LIN {X 0,Y 284.126,Z 570.884,A -85,B 0,C 180,E1 -16986.134,E2 -16986.134} C_VEL
LIN {X 0,Y 285.514,Z 585.301,A -85,B 0,C 180,E1 -16986.902,E2 -16986.902} C_VEL
LIN {X 0,Y 286.444,Z 597.974,A -85,B 0,C 180,E1 -16987.838,E2 -16987.838} C_VEL
LIN {X 0,Y 287.043,Z 610.993,A -85,B 0,C 180,E1 -16989.097,E2 -16989.097} C_VEL
LIN {X 0,Y 287.237,Z 622.835,A -85,B 0,C 180,E1 -16990.527,E2 -16990.527} C_VEL
LIN {X 0,Y 286.97,Z 632.757,A -85,B 0,C 180,E1 -16991.99,E2 -16991.99} C_VEL
LIN {X 0,Y 285.776,Z 641.656,A -85,B 0,C 180,E1 -16993.56,E2 -16993.56} C_VEL
LIN {X 0,Y 284.464,Z 651.441,A -85,B 0,C 180,E1 -16995.696,E2 -16995.696} C_VEL
LIN {X 0,Y 283.789,Z 659.297,A -85,B 0,C 180,E1 -16997.848,E2 -16997.848} C_VEL
LIN {X 0,Y 283.448,Z 665.562,A -85,B 0,C 180,E1 -17000.005,E2 -17000.005} C_VEL
LIN {X 0,Y 283.441,Z 670.658,A -85,B 0,C 180,E1 -17002.234,E2 -17002.234} C_VEL
LIN {X 0,Y 283.67,Z 674.283,A -85,B 0,C 180,E1 -17004.313,E2 -17004.313} C_VEL
LIN {X 0,Y 283.832,Z 676.171,A -85,B 0,C 180,E1 -17005.74,E2 -17005.74} C_VEL
LIN {X 0,Y 283.974,Z 677.598,A -85,B 0,C 180,E1 -17007.163,E2 -17007.163} C_VEL
LIN {X 0,Y 284.233,Z 678.549,A -85,B 0,C 180,E1 -17008.583,E2 -17008.583} C_VEL
LIN {X 0,Y 284.459,Z 679.061,A -85,B 0,C 180,E1 -17010,E2 -17010} C_VEL
LIN {X 0,Y 283.861,Z 678.655,A -85,B 0,C 180,E1 -17012.838,E2 -17012.838} C_VEL
LIN {X 0,Y 283.692,Z 677.798,A -85,B 0,C 180,E1 -17014.262,E2 -17014.262} C_VEL
LIN {X 0,Y 283.264,Z 674.815,A -85,B 0,C 180,E1 -17017.126,E2 -17017.126} C_VEL
LIN {X 0,Y 283.136,Z 671.429,A -85,B 0,C 180,E1 -17019.285,E2 -17019.285} C_VEL
LIN {X 0,Y 283.389,Z 667.023,A -85,B 0,C 180,E1 -17021.444,E2 -17021.444} C_VEL
LIN {X 0,Y 284.212,Z 660.522,A -85,B 0,C 180,E1 -17023.952,E2 -17023.952} C_VEL
LIN {X 0,Y 285.074,Z 654.806,A -85,B 0,C 180,E1 -17025.735,E2 -17025.735} C_VEL
LIN {X 0,Y 286.836,Z 646.656,A -85,B 0,C 180,E1 -17027.835,E2 -17027.835} C_VEL
LIN {X 0,Y 289.074,Z 636.649,A -85,B 0,C 180,E1 -17029.9,E2 -17029.9} C_VEL
LIN {X 0,Y 290.359,Z 625.448,A -85,B 0,C 180,E1 -17031.848,E2 -17031.848} C_VEL
LIN {X 0,Y 291.533,Z 612.796,A -85,B 0,C 180,E1 -17033.642,E2 -17033.642} C_VEL
LIN {X 0,Y 291.696,Z 600.649,A -85,B 0,C 180,E1 -17035.122,E2 -17035.122} C_VEL
LIN {X 0,Y 290.667,Z 587.531,A -85,B 0,C 180,E1 -17036.541,E2 -17036.541} C_VEL
LIN {X 0,Y 288.705,Z 574.355,A -85,B 0,C 180,E1 -17037.828,E2 -17037.828} C_VEL
LIN {X 0,Y 286.15,Z 563.427,A -85,B 0,C 180,E1 -17038.838,E2 -17038.838} C_VEL
LIN {X 0,Y 285.515,Z 560.161,A -85,B 0,C 180,E1 -17039.106,E2 -17039.106} C_VEL
LIN {X 0,Y 287.109,Z 549.67,A -85,B 0,C 180,E1 -17043.667,E2 -17043.667} C_VEL
LIN {X 0,Y 289.085,Z 539.77,A -85,B 0,C 180,E1 -17048.193,E2 -17048.193} C_VEL
LIN {X 0,Y 289.175,Z 537.775,A -85,B 0,C 180,E1 -17049.191,E2 -17049.191} C_VEL
LIN {X 0,Y 288.339,Z 532.571,A -85,B 0,C 180,E1 -17052.035,E2 -17052.035} C_VEL
LIN {X 0,Y 287.355,Z 527.335,A -85,B 0,C 180,E1 -17055.176,E2 -17055.176} C_VEL
LIN {X 0,Y 286.33,Z 522.347,A -85,B 0,C 180,E1 -17058.493,E2 -17058.493} C_VEL
LIN {X 0,Y 285.335,Z 517.677,A -85,B 0,C 180,E1 -17062.017,E2 -17062.017} C_VEL
LIN {X 0,Y 284.314,Z 513.065,A -85,B 0,C 180,E1 -17066.208,E2 -17066.208} C_VEL
LIN {X 0,Y 284.361,Z 513.057,A -85,B 0,C 180,E1 -17070.377,E2 -17070.377} C_VEL
LIN {X 0,Y 284.381,Z 513.053,A -85,B 0,C 180,E1 -17073.587,E2 -17073.587} C_VEL
LIN {X 0,Y 284.369,Z 513.056,A -85,B 0,C 180,E1 -17076.707,E2 -17076.707} C_VEL
LIN {X 0,Y 284.406,Z 513.055,A -85,B 0,C 180,E1 -17081.262,E2 -17081.262} C_VEL
LIN {X 0,Y 284.495,Z 513.044,A -85,B 0,C 180,E1 -17084.459,E2 -17084.459} C_VEL
LIN {X 0,Y 284.492,Z 513.04,A -85,B 0,C 180,E1 -17088.602,E2 -17088.602} C_VEL
LIN {X 0,Y 284.663,Z 513.019,A -85,B 0,C 180,E1 -17091.482,E2 -17091.482} C_VEL
LIN {X 0,Y 284.6,Z 513.031,A -85,B 0,C 180,E1 -17094.332,E2 -17094.332} C_VEL
LIN {X 0,Y 284.854,Z 513.002,A -85,B 0,C 180,E1 -17098.587,E2 -17098.587} C_VEL
LIN {X 0,Y 284.858,Z 513.003,A -85,B 0,C 180,E1 -17101.414,E2 -17101.414} C_VEL
LIN {X 0,Y 284.582,Z 513.031,A -85,B 0,C 180,E1 -17105.536,E2 -17105.536} C_VEL
LIN {X 0,Y 285.22,Z 515.176,A -85,B 0,C 180,E1 -17105.834,E2 -17105.834} C_VEL
LIN {X 0,Y 288.767,Z 521.378,A -85,B 0,C 180,E1 -17106.99,E2 -17106.99} C_VEL
LIN {X 0,Y 293.537,Z 532.381,A -85,B 0,C 180,E1 -17108.954,E2 -17108.954} C_VEL
LIN {X 0,Y 296.554,Z 541.172,A -85,B 0,C 180,E1 -17110.584,E2 -17110.584} C_VEL
LIN {X 0,Y 298.373,Z 548.706,A -85,B 0,C 180,E1 -17112.039,E2 -17112.039} C_VEL
LIN {X 0,Y 297.747,Z 553.329,A -85,B 0,C 180,E1 -17112.77,E2 -17112.77} C_VEL
LIN {X 0,Y 295.774,Z 562.817,A -85,B 0,C 180,E1 -17114.447,E2 -17114.447} C_VEL
LIN {X 0,Y 293.677,Z 571.656,A -85,B 0,C 180,E1 -17116.417,E2 -17116.417} C_VEL
LIN {X 0,Y 291.671,Z 579.309,A -85,B 0,C 180,E1 -17118.563,E2 -17118.563} C_VEL
LIN {X 0,Y 290.018,Z 584.973,A -85,B 0,C 180,E1 -17120.572,E2 -17120.572} C_VEL
LIN {X 0,Y 288.412,Z 590.115,A -85,B 0,C 180,E1 -17122.948,E2 -17122.948} C_VEL
LIN {X 0,Y 287.211,Z 593.585,A -85,B 0,C 180,E1 -17125.124,E2 -17125.124} C_VEL
LIN {X 0,Y 286.03,Z 596.426,A -85,B 0,C 180,E1 -17127.83,E2 -17127.83} C_VEL
LIN {X 0,Y 285.27,Z 597.703,A -85,B 0,C 180,E1 -17130.427,E2 -17130.427} C_VEL
LIN {X 0,Y 284.803,Z 597.654,A -85,B 0,C 180,E1 -17132.964,E2 -17132.964} C_VEL
LIN {X 0,Y 284.628,Z 596.402,A -85,B 0,C 180,E1 -17135.429,E2 -17135.429} C_VEL
LIN {X 0,Y 284.722,Z 593.682,A -85,B 0,C 180,E1 -17138.105,E2 -17138.105} C_VEL
LIN {X 0,Y 285.201,Z 589.25,A -85,B 0,C 180,E1 -17140.843,E2 -17140.843} C_VEL
LIN {X 0,Y 285.807,Z 584.791,A -85,B 0,C 180,E1 -17142.886,E2 -17142.886} C_VEL
LIN {X 0,Y 286.656,Z 578.043,A -85,B 0,C 180,E1 -17145.317,E2 -17145.317} C_VEL
LIN {X 0,Y 287.491,Z 571.602,A -85,B 0,C 180,E1 -17147.171,E2 -17147.171} C_VEL
LIN {X 0,Y 288.739,Z 562.674,A -85,B 0,C 180,E1 -17149.253,E2 -17149.253} C_VEL
LIN {X 0,Y 289.919,Z 552.701,A -85,B 0,C 180,E1 -17151.147,E2 -17151.147} C_VEL
LIN {X 0,Y 291.151,Z 541.755,A -85,B 0,C 180,E1 -17152.806,E2 -17152.806} C_VEL
LIN {X 0,Y 291.404,Z 537.676,A -85,B 0,C 180,E1 -17153.35,E2 -17153.35} C_VEL
LIN {X 0,Y 288.411,Z 526.574,A -85,B 0,C 180,E1 -17154.868,E2 -17154.868} C_VEL
LIN {X 0,Y 284.684,Z 514.526,A -85,B 0,C 180,E1 -17156.257,E2 -17156.257} C_VEL
LIN {X 0,Y 284.32,Z 513.07,A -85,B 0,C 180,E1 -17156.421,E2 -17156.421} C_VEL
LIN {X 0,Y 284.364,Z 513.063,A -85,B 0,C 180,E1 -17160.376,E2 -17160.376} C_VEL
LIN {X 0,Y 284.385,Z 513.062,A -85,B 0,C 180,E1 -17163.587,E2 -17163.587} C_VEL
LIN {X 0,Y 284.337,Z 513.065,A -85,B 0,C 180,E1 -17166.704,E2 -17166.704} C_VEL
LIN {X 0,Y 284.381,Z 513.06,A -85,B 0,C 180,E1 -17169.904,E2 -17169.904} C_VEL
LIN {X 0,Y 284.452,Z 513.05,A -85,B 0,C 180,E1 -17174.492,E2 -17174.492} C_VEL
LIN {X 0,Y 284.488,Z 513.046,A -85,B 0,C 180,E1 -17178.601,E2 -17178.601} C_VEL
LIN {X 0,Y 284.613,Z 513.033,A -85,B 0,C 180,E1 -17181.48,E2 -17181.48} C_VEL
LIN {X 0,Y 284.581,Z 513.034,A -85,B 0,C 180,E1 -17184.331,E2 -17184.331} C_VEL
LIN {X 0,Y 284.855,Z 513,A -85,B 0,C 180,E1 -17188.586,E2 -17188.586} C_VEL
LIN {X 0,Y 284.857,Z 513.003,A -85,B 0,C 180,E1 -17191.414,E2 -17191.414} C_VEL
LIN {X 0,Y 284.648,Z 513.029,A -85,B 0,C 180,E1 -17197.091,E2 -17197.091} C_VEL
LIN {X 0,Y 284.518,Z 513.041,A -85,B 0,C 180,E1 -17199.957,E2 -17199.957} C_VEL
LIN {X 0,Y 284.468,Z 513.048,A -85,B 0,C 180,E1 -17204.303,E2 -17204.303} C_VEL
LIN {X 0,Y 284.39,Z 513.058,A -85,B 0,C 180,E1 -17208.739,E2 -17208.739} C_VEL
LIN {X 0,Y 284.33,Z 513.066,A -85,B 0,C 180,E1 -17211.763,E2 -17211.763} C_VEL
LIN {X 0,Y 284.32,Z 513.068,A -85,B 0,C 180,E1 -17214.848,E2 -17214.848} C_VEL
LIN {X 0,Y 284.295,Z 513.069,A -85,B 0,C 180,E1 -17218.014,E2 -17218.014} C_VEL
LIN {X 0,Y 284.29,Z 513.074,A -85,B 0,C 180,E1 -17221.275,E2 -17221.275} C_VEL
LIN {X 0,Y 284.339,Z 513.066,A -85,B 0,C 180,E1 -17225.346,E2 -17225.346} C_VEL
LIN {X 0,Y 284.304,Z 513.068,A -85,B 0,C 180,E1 -17228.17,E2 -17228.17} C_VEL
LIN {X 0,Y 284.24,Z 513.075,A -85,B 0,C 180,E1 -17232.117,E2 -17232.117} C_VEL
LIN {X 0,Y 284.257,Z 513.074,A -85,B 0,C 180,E1 -17236.189,E2 -17236.189} C_VEL
LIN {X 0,Y 284.309,Z 513.067,A -85,B 0,C 180,E1 -17240.024,E2 -17240.024} C_VEL
LIN {X 0,Y 284.333,Z 513.065,A -85,B 0,C 180,E1 -17243.613,E2 -17243.613} C_VEL
LIN {X 0,Y 284.31,Z 513.071,A -85,B 0,C 180,E1 -17247.189,E2 -17247.189} C_VEL
LIN {X 0,Y 284.361,Z 513.06,A -85,B 0,C 180,E1 -17250.376,E2 -17250.376} C_VEL
LIN {X 0,Y 284.38,Z 513.06,A -85,B 0,C 180,E1 -17253.586,E2 -17253.586} C_VEL
LIN {X 0,Y 284.335,Z 513.067,A -85,B 0,C 180,E1 -17256.704,E2 -17256.704} C_VEL
LIN {X 0,Y 284.406,Z 513.058,A -85,B 0,C 180,E1 -17261.261,E2 -17261.261} C_VEL
LIN {X 0,Y 284.494,Z 513.046,A -85,B 0,C 180,E1 -17264.459,E2 -17264.459} C_VEL
LIN {X 0,Y 284.485,Z 513.047,A -85,B 0,C 180,E1 -17268.601,E2 -17268.601} C_VEL
LIN {X 0,Y 284.613,Z 513.031,A -85,B 0,C 180,E1 -17271.479,E2 -17271.479} C_VEL
LIN {X 0,Y 284.58,Z 513.034,A -85,B 0,C 180,E1 -17274.33,E2 -17274.33} C_VEL
LIN {X 0,Y 284.853,Z 513.002,A -85,B 0,C 180,E1 -17278.586,E2 -17278.586} C_VEL
LIN {X 0,Y 284.853,Z 513.001,A -85,B 0,C 180,E1 -17281.413,E2 -17281.413} C_VEL
LIN {X 0,Y 284.634,Z 513.029,A -85,B 0,C 180,E1 -17287.222,E2 -17287.222} C_VEL
LIN {X 0,Y 284.519,Z 513.041,A -85,B 0,C 180,E1 -17289.957,E2 -17289.957} C_VEL
LIN {X 0,Y 284.452,Z 513.049,A -85,B 0,C 180,E1 -17293.37,E2 -17293.37} C_VEL
LIN {X 0,Y 283.765,Z 513.138,A -85,B 0,C 180,E1 -17294.551,E2 -17294.551} C_VEL
LIN {X 0,Y 280.888,Z 513.496,A -85,B 0,C 180,E1 -17296.474,E2 -17296.474} C_VEL
LIN {X 0,Y 278.45,Z 513.799,A -85,B 0,C 180,E1 -17298.036,E2 -17298.036} C_VEL
LIN {X 0,Y 277.398,Z 513.93,A -85,B 0,C 180,E1 -17299.247,E2 -17299.247} C_VEL
LIN {X 0,Y 277.308,Z 513.939,A -85,B 0,C 180,E1 -17299.657,E2 -17299.657} C_VEL
LIN {X 0,Y 277.282,Z 513.943,A -85,B 0,C 180,E1 -17304.152,E2 -17304.152} C_VEL
LIN {X 0,Y 277.274,Z 513.944,A -85,B 0,C 180,E1 -17307.484,E2 -17307.484} C_VEL
LIN {X 0,Y 277.248,Z 513.949,A -85,B 0,C 180,E1 -17310.472,E2 -17310.472} C_VEL
LIN {X 0,Y 277.247,Z 513.948,A -85,B 0,C 180,E1 -17313.896,E2 -17313.896} C_VEL
LIN {X 0,Y 277.268,Z 513.946,A -85,B 0,C 180,E1 -17317.469,E2 -17317.469} C_VEL
LIN {X 0,Y 277.302,Z 514.049,A -85,B 0,C 180,E1 -17319.647,E2 -17319.647} C_VEL
LIN {X 0,Y 278.816,Z 521.939,A -85,B 0,C 180,E1 -17323.881,E2 -17323.881} C_VEL
LIN {X 0,Y 280.369,Z 529.967,A -85,B 0,C 180,E1 -17327.953,E2 -17327.953} C_VEL
LIN {X 0,Y 281.482,Z 535.685,A -85,B 0,C 180,E1 -17330.715,E2 -17330.715} C_VEL
LIN {X 0,Y 281.516,Z 539.122,A -85,B 0,C 180,E1 -17332.293,E2 -17332.293} C_VEL
LIN {X 0,Y 279.904,Z 548.574,A -85,B 0,C 180,E1 -17336.469,E2 -17336.469} C_VEL
LIN {X 0,Y 278.223,Z 559.738,A -85,B 0,C 180,E1 -17341.318,E2 -17341.318} C_VEL
LIN {X 0,Y 277.139,Z 570.066,A -85,B 0,C 180,E1 -17345.685,E2 -17345.685} C_VEL
LIN {X 0,Y 278.508,Z 584.506,A -85,B 0,C 180,E1 -17346.483,E2 -17346.483} C_VEL
LIN {X 0,Y 279.487,Z 598.226,A -85,B 0,C 180,E1 -17347.548,E2 -17347.548} C_VEL
LIN {X 0,Y 280.052,Z 611.206,A -85,B 0,C 180,E1 -17348.858,E2 -17348.858} C_VEL
LIN {X 0,Y 280.184,Z 623.313,A -85,B 0,C 180,E1 -17350.398,E2 -17350.398} C_VEL
LIN {X 0,Y 280.017,Z 631.921,A -85,B 0,C 180,E1 -17351.716,E2 -17351.716} C_VEL
LIN {X 0,Y 278.804,Z 640.734,A -85,B 0,C 180,E1 -17353.314,E2 -17353.314} C_VEL
LIN {X 0,Y 277.518,Z 649.792,A -85,B 0,C 180,E1 -17355.331,E2 -17355.331} C_VEL
LIN {X 0,Y 276.896,Z 656.55,A -85,B 0,C 180,E1 -17357.168,E2 -17357.168} C_VEL
LIN {X 0,Y 276.492,Z 662.166,A -85,B 0,C 180,E1 -17359.01,E2 -17359.01} C_VEL
LIN {X 0,Y 276.354,Z 667.634,A -85,B 0,C 180,E1 -17361.223,E2 -17361.223} C_VEL
LIN {X 0,Y 276.507,Z 671.865,A -85,B 0,C 180,E1 -17363.432,E2 -17363.432} C_VEL
LIN {X 0,Y 276.787,Z 674.949,A -85,B 0,C 180,E1 -17365.631,E2 -17365.631} C_VEL
LIN {X 0,Y 276.937,Z 676.414,A -85,B 0,C 180,E1 -17367.091,E2 -17367.091} C_VEL
LIN {X 0,Y 277.214,Z 677.425,A -85,B 0,C 180,E1 -17368.547,E2 -17368.547} C_VEL
LIN {X 0,Y 277.441,Z 677.967,A -85,B 0,C 180,E1 -17370,E2 -17370} C_VEL
LIN {X 0,Y 276.809,Z 677.621,A -85,B 0,C 180,E1 -17372.911,E2 -17372.911} C_VEL
LIN {X 0,Y 276.606,Z 676.814,A -85,B 0,C 180,E1 -17374.372,E2 -17374.372} C_VEL
LIN {X 0,Y 276.177,Z 673.883,A -85,B 0,C 180,E1 -17377.31,E2 -17377.31} C_VEL
LIN {X 0,Y 276.078,Z 670.565,A -85,B 0,C 180,E1 -17379.525,E2 -17379.525} C_VEL
LIN {X 0,Y 276.37,Z 666.254,A -85,B 0,C 180,E1 -17381.738,E2 -17381.738} C_VEL
LIN {X 0,Y 277.265,Z 659.85,A -85,B 0,C 180,E1 -17384.309,E2 -17384.309} C_VEL
LIN {X 0,Y 278.7,Z 651.977,A -85,B 0,C 180,E1 -17386.783,E2 -17386.783} C_VEL
LIN {X 0,Y 280.714,Z 643.129,A -85,B 0,C 180,E1 -17388.994,E2 -17388.994} C_VEL
LIN {X 0,Y 282.339,Z 636.416,A -85,B 0,C 180,E1 -17390.395,E2 -17390.395} C_VEL
LIN {X 0,Y 283.731,Z 625.469,A -85,B 0,C 180,E1 -17392.386,E2 -17392.386} C_VEL
LIN {X 0,Y 284.978,Z 613.667,A -85,B 0,C 180,E1 -17394.15,E2 -17394.15} C_VEL
LIN {X 0,Y 285.253,Z 601.377,A -85,B 0,C 180,E1 -17395.737,E2 -17395.737} C_VEL
LIN {X 0,Y 284.452,Z 588.865,A -85,B 0,C 180,E1 -17397.195,E2 -17397.195} C_VEL
LIN {X 0,Y 282.831,Z 576.714,A -85,B 0,C 180,E1 -17398.47,E2 -17398.47} C_VEL
LIN {X 0,Y 279.839,Z 562.965,A -85,B 0,C 180,E1 -17399.848,E2 -17399.848} C_VEL
LIN {X 0,Y 278.851,Z 558.99,A -85,B 0,C 180,E1 -17400.218,E2 -17400.218} C_VEL
LIN {X 0,Y 278.829,Z 558.603,A -85,B 0,C 180,E1 -17400.273,E2 -17400.273} C_VEL
LIN {X 0,Y 280.69,Z 547.821,A -85,B 0,C 180,E1 -17405.162,E2 -17405.162} C_VEL
LIN {X 0,Y 282.19,Z 540.774,A -85,B 0,C 180,E1 -17408.509,E2 -17408.509} C_VEL
LIN {X 0,Y 281.944,Z 537.239,A -85,B 0,C 180,E1 -17410.399,E2 -17410.399} C_VEL
LIN {X 0,Y 280.753,Z 530.313,A -85,B 0,C 180,E1 -17414.501,E2 -17414.501} C_VEL
LIN {X 0,Y 279.61,Z 524.759,A -85,B 0,C 180,E1 -17418.236,E2 -17418.236} C_VEL
LIN {X 0,Y 278.727,Z 520.574,A -85,B 0,C 180,E1 -17421.413,E2 -17421.413} C_VEL
LIN {X 0,Y 277.959,Z 517.056,A -85,B 0,C 180,E1 -17424.441,E2 -17424.441} C_VEL
LIN {X 0,Y 277.245,Z 513.946,A -85,B 0,C 180,E1 -17427.554,E2 -17427.554} C_VEL
LIN {X 0,Y 277.274,Z 513.94,A -85,B 0,C 180,E1 -17431.211,E2 -17431.211} C_VEL
LIN {X 0,Y 277.317,Z 513.939,A -85,B 0,C 180,E1 -17434.48,E2 -17434.48} C_VEL
LIN {X 0,Y 277.288,Z 513.944,A -85,B 0,C 180,E1 -17437.655,E2 -17437.655} C_VEL
LIN {X 0,Y 277.348,Z 513.938,A -85,B 0,C 180,E1 -17440.767,E2 -17440.767} C_VEL
LIN {X 0,Y 277.438,Z 513.918,A -85,B 0,C 180,E1 -17445.326,E2 -17445.326} C_VEL
LIN {X 0,Y 277.51,Z 513.916,A -85,B 0,C 180,E1 -17449.789,E2 -17449.789} C_VEL
LIN {X 0,Y 277.657,Z 513.894,A -85,B 0,C 180,E1 -17452.73,E2 -17452.73} C_VEL
LIN {X 0,Y 277.82,Z 513.878,A -85,B 0,C 180,E1 -17458.551,E2 -17458.551} C_VEL
LIN {X 0,Y 277.824,Z 513.879,A -85,B 0,C 180,E1 -17461.45,E2 -17461.45} C_VEL
LIN {X 0,Y 277.471,Z 514.008,A -85,B 0,C 180,E1 -17464.313,E2 -17464.313} C_VEL
LIN {X 0,Y 278.396,Z 516.611,A -85,B 0,C 180,E1 -17464.707,E2 -17464.707} C_VEL
LIN {X 0,Y 279.52,Z 518.046,A -85,B 0,C 180,E1 -17465.049,E2 -17465.049} C_VEL
LIN {X 0,Y 284.001,Z 526.61,A -85,B 0,C 180,E1 -17466.715,E2 -17466.715} C_VEL
LIN {X 0,Y 287.682,Z 535.557,A -85,B 0,C 180,E1 -17468.429,E2 -17468.429} C_VEL
LIN {X 0,Y 290.745,Z 545.046,A -85,B 0,C 180,E1 -17470.303,E2 -17470.303} C_VEL
LIN {X 0,Y 292.041,Z 550.664,A -85,B 0,C 180,E1 -17471.452,E2 -17471.452} C_VEL
LIN {X 0,Y 291.793,Z 553.762,A -85,B 0,C 180,E1 -17471.99,E2 -17471.99} C_VEL
LIN {X 0,Y 289.515,Z 564.005,A -85,B 0,C 180,E1 -17473.83,E2 -17473.83} C_VEL
LIN {X 0,Y 287.235,Z 573.052,A -85,B 0,C 180,E1 -17475.894,E2 -17475.894} C_VEL
LIN {X 0,Y 285.251,Z 580.192,A -85,B 0,C 180,E1 -17477.938,E2 -17477.938} C_VEL
LIN {X 0,Y 283.229,Z 586.715,A -85,B 0,C 180,E1 -17480.329,E2 -17480.329} C_VEL
LIN {X 0,Y 281.664,Z 591.393,A -85,B 0,C 180,E1 -17482.598,E2 -17482.598} C_VEL
LIN {X 0,Y 280.102,Z 595.529,A -85,B 0,C 180,E1 -17485.408,E2 -17485.408} C_VEL
LIN {X 0,Y 278.932,Z 597.926,A -85,B 0,C 180,E1 -17488.131,E2 -17488.131} C_VEL
LIN {X 0,Y 278.165,Z 598.89,A -85,B 0,C 180,E1 -17490.791,E2 -17490.791} C_VEL
LIN {X 0,Y 277.756,Z 598.557,A -85,B 0,C 180,E1 -17493.384,E2 -17493.384} C_VEL
LIN {X 0,Y 277.596,Z 597.016,A -85,B 0,C 180,E1 -17495.888,E2 -17495.888} C_VEL
LIN {X 0,Y 277.699,Z 594.36,A -85,B 0,C 180,E1 -17498.32,E2 -17498.32} C_VEL
LIN {X 0,Y 278.223,Z 589.923,A -85,B 0,C 180,E1 -17501.055,E2 -17501.055} C_VEL
LIN {X 0,Y 278.934,Z 584.846,A -85,B 0,C 180,E1 -17503.364,E2 -17503.364} C_VEL
LIN {X 0,Y 279.847,Z 577.599,A -85,B 0,C 180,E1 -17505.906,E2 -17505.906} C_VEL
LIN {X 0,Y 281.041,Z 569.082,A -85,B 0,C 180,E1 -17508.254,E2 -17508.254} C_VEL
LIN {X 0,Y 282.22,Z 560.059,A -85,B 0,C 180,E1 -17510.236,E2 -17510.236} C_VEL
LIN {X 0,Y 283.379,Z 550.663,A -85,B 0,C 180,E1 -17511.928,E2 -17511.928} C_VEL
LIN {X 0,Y 284.446,Z 541.032,A -85,B 0,C 180,E1 -17513.359,E2 -17513.359} C_VEL
LIN {X 0,Y 284.474,Z 539.04,A -85,B 0,C 180,E1 -17513.635,E2 -17513.635} C_VEL
LIN {X 0,Y 281.569,Z 528.059,A -85,B 0,C 180,E1 -17515.182,E2 -17515.182} C_VEL
LIN {X 0,Y 277.926,Z 516.211,A -85,B 0,C 180,E1 -17516.592,E2 -17516.592} C_VEL
LIN {X 0,Y 277.281,Z 513.948,A -85,B 0,C 180,E1 -17516.848,E2 -17516.848} C_VEL
LIN {X 0,Y 277.296,Z 513.947,A -85,B 0,C 180,E1 -17521.213,E2 -17521.213} C_VEL
LIN {X 0,Y 277.316,Z 513.94,A -85,B 0,C 180,E1 -17524.479,E2 -17524.479} C_VEL
LIN {X 0,Y 277.271,Z 513.947,A -85,B 0,C 180,E1 -17527.653,E2 -17527.653} C_VEL
LIN {X 0,Y 277.329,Z 513.938,A -85,B 0,C 180,E1 -17530.765,E2 -17530.765} C_VEL
LIN {X 0,Y 277.414,Z 513.932,A -85,B 0,C 180,E1 -17535.325,E2 -17535.325} C_VEL
LIN {X 0,Y 277.462,Z 513.922,A -85,B 0,C 180,E1 -17539.787,E2 -17539.787} C_VEL
LIN {X 0,Y 277.606,Z 513.903,A -85,B 0,C 180,E1 -17542.728,E2 -17542.728} C_VEL
LIN {X 0,Y 277.701,Z 513.894,A -85,B 0,C 180,E1 -17547.098,E2 -17547.098} C_VEL
LIN {X 0,Y 277.849,Z 513.873,A -85,B 0,C 180,E1 -17550,E2 -17550} C_VEL
LIN {X 0,Y 277.697,Z 513.893,A -85,B 0,C 180,E1 -17552.901,E2 -17552.901} C_VEL
LIN {X 0,Y 277.606,Z 513.906,A -85,B 0,C 180,E1 -17557.272,E2 -17557.272} C_VEL
LIN {X 0,Y 277.462,Z 513.92,A -85,B 0,C 180,E1 -17560.213,E2 -17560.213} C_VEL
LIN {X 0,Y 277.414,Z 513.927,A -85,B 0,C 180,E1 -17564.675,E2 -17564.675} C_VEL
LIN {X 0,Y 277.339,Z 513.94,A -85,B 0,C 180,E1 -17569.234,E2 -17569.234} C_VEL
LIN {X 0,Y 277.292,Z 513.941,A -85,B 0,C 180,E1 -17573.924,E2 -17573.924} C_VEL
LIN {X 0,Y 277.285,Z 513.945,A -85,B 0,C 180,E1 -17577.487,E2 -17577.487} C_VEL
LIN {X 0,Y 277.251,Z 513.947,A -85,B 0,C 180,E1 -17580.472,E2 -17580.472} C_VEL
LIN {X 0,Y 277.249,Z 513.946,A -85,B 0,C 180,E1 -17583.895,E2 -17583.895} C_VEL
LIN {X 0,Y 277.263,Z 513.947,A -85,B 0,C 180,E1 -17587.47,E2 -17587.47} C_VEL
LIN {X 0,Y 277.187,Z 513.958,A -85,B 0,C 180,E1 -17591.241,E2 -17591.241} C_VEL
LIN {X 0,Y 277.203,Z 513.957,A -85,B 0,C 180,E1 -17595.226,E2 -17595.226} C_VEL
LIN {X 0,Y 277.225,Z 513.951,A -85,B 0,C 180,E1 -17599.512,E2 -17599.512} C_VEL
LIN {X 0,Y 277.267,Z 513.944,A -85,B 0,C 180,E1 -17602.53,E2 -17602.53} C_VEL
LIN {X 0,Y 277.249,Z 513.947,A -85,B 0,C 180,E1 -17606.104,E2 -17606.104} C_VEL
LIN {X 0,Y 277.264,Z 513.945,A -85,B 0,C 180,E1 -17609.538,E2 -17609.538} C_VEL
LIN {X 0,Y 277.361,Z 513.936,A -85,B 0,C 180,E1 -17612.864,E2 -17612.864} C_VEL
LIN {X 0,Y 277.299,Z 513.94,A -85,B 0,C 180,E1 -17616.076,E2 -17616.076} C_VEL
LIN {X 0,Y 277.347,Z 513.937,A -85,B 0,C 180,E1 -17620.766,E2 -17620.766} C_VEL
LIN {X 0,Y 277.437,Z 513.925,A -85,B 0,C 180,E1 -17625.326,E2 -17625.326} C_VEL
LIN {X 0,Y 277.459,Z 513.921,A -85,B 0,C 180,E1 -17629.786,E2 -17629.786} C_VEL
LIN {X 0,Y 277.607,Z 513.906,A -85,B 0,C 180,E1 -17632.727,E2 -17632.727} C_VEL
LIN {X 0,Y 277.82,Z 513.878,A -85,B 0,C 180,E1 -17638.55,E2 -17638.55} C_VEL
LIN {X 0,Y 277.819,Z 513.877,A -85,B 0,C 180,E1 -17641.449,E2 -17641.449} C_VEL
LIN {X 0,Y 277.603,Z 513.905,A -85,B 0,C 180,E1 -17647.272,E2 -17647.272} C_VEL
LIN {X 0,Y 277.462,Z 513.921,A -85,B 0,C 180,E1 -17650.213,E2 -17650.213} C_VEL
LIN {X 0,Y 277.411,Z 513.929,A -85,B 0,C 180,E1 -17654.675,E2 -17654.675} C_VEL
LIN {X 0,Y 277.325,Z 513.939,A -85,B 0,C 180,E1 -17659.235,E2 -17659.235} C_VEL
LIN {X 0,Y 277.308,Z 513.939,A -85,B 0,C 180,E1 -17659.657,E2 -17659.657} C_VEL
LIN {X 0,Y 276.615,Z 514.029,A -85,B 0,C 180,E1 -17660.868,E2 -17660.868} C_VEL
LIN {X 0,Y 273.71,Z 514.391,A -85,B 0,C 180,E1 -17662.84,E2 -17662.84} C_VEL
LIN {X 0,Y 271.277,Z 514.693,A -85,B 0,C 180,E1 -17664.443,E2 -17664.443} C_VEL
LIN {X 0,Y 270.266,Z 514.817,A -85,B 0,C 180,E1 -17665.687,E2 -17665.687} C_VEL
LIN {X 0,Y 270.201,Z 514.825,A -85,B 0,C 180,E1 -17666.108,E2 -17666.108} C_VEL
LIN {X 0,Y 270.185,Z 514.827,A -85,B 0,C 180,E1 -17669.618,E2 -17669.618} C_VEL
LIN {X 0,Y 270.215,Z 514.824,A -85,B 0,C 180,E1 -17673.666,E2 -17673.666} C_VEL
LIN {X 0,Y 270.218,Z 514.827,A -85,B 0,C 180,E1 -17676.741,E2 -17676.741} C_VEL
LIN {X 0,Y 270.231,Z 514.861,A -85,B 0,C 180,E1 -17679.219,E2 -17679.219} C_VEL
LIN {X 0,Y 271.779,Z 522.824,A -85,B 0,C 180,E1 -17683.609,E2 -17683.609} C_VEL
LIN {X 0,Y 273.074,Z 529.533,A -85,B 0,C 180,E1 -17687.116,E2 -17687.116} C_VEL
LIN {X 0,Y 274.309,Z 535.766,A -85,B 0,C 180,E1 -17690.23,E2 -17690.23} C_VEL
LIN {X 0,Y 274.595,Z 537.754,A -85,B 0,C 180,E1 -17691.197,E2 -17691.197} C_VEL
LIN {X 0,Y 274.043,Z 542.089,A -85,B 0,C 180,E1 -17693.203,E2 -17693.203} C_VEL
LIN {X 0,Y 272.516,Z 550.994,A -85,B 0,C 180,E1 -17697.209,E2 -17697.209} C_VEL
LIN {X 0,Y 270.893,Z 562.06,A -85,B 0,C 180,E1 -17702.161,E2 -17702.161} C_VEL
LIN {X 0,Y 270.132,Z 568.915,A -85,B 0,C 180,E1 -17705.193,E2 -17705.193} C_VEL
LIN {X 0,Y 271.532,Z 583.773,A -85,B 0,C 180,E1 -17706.048,E2 -17706.048} C_VEL
LIN {X 0,Y 272.405,Z 596.261,A -85,B 0,C 180,E1 -17707.037,E2 -17707.037} C_VEL
LIN {X 0,Y 273.012,Z 609.745,A -85,B 0,C 180,E1 -17708.424,E2 -17708.424} C_VEL
LIN {X 0,Y 273.131,Z 621.035,A -85,B 0,C 180,E1 -17709.87,E2 -17709.87} C_VEL
LIN {X 0,Y 272.917,Z 632.052,A -85,B 0,C 180,E1 -17711.612,E2 -17711.612} C_VEL
LIN {X 0,Y 271.581,Z 641.676,A -85,B 0,C 180,E1 -17713.462,E2 -17713.462} C_VEL
LIN {X 0,Y 270.429,Z 649.579,A -85,B 0,C 180,E1 -17715.322,E2 -17715.322} C_VEL
LIN {X 0,Y 269.799,Z 656.196,A -85,B 0,C 180,E1 -17717.208,E2 -17717.208} C_VEL
LIN {X 0,Y 269.367,Z 662.696,A -85,B 0,C 180,E1 -17719.477,E2 -17719.477} C_VEL
LIN {X 0,Y 269.329,Z 667.969,A -85,B 0,C 180,E1 -17721.824,E2 -17721.824} C_VEL
LIN {X 0,Y 269.574,Z 671.754,A -85,B 0,C 180,E1 -17724.014,E2 -17724.014} C_VEL
LIN {X 0,Y 269.744,Z 673.716,A -85,B 0,C 180,E1 -17725.517,E2 -17725.517} C_VEL
LIN {X 0,Y 269.9,Z 675.215,A -85,B 0,C 180,E1 -17727.015,E2 -17727.015} C_VEL
LIN {X 0,Y 270.192,Z 676.291,A -85,B 0,C 180,E1 -17728.51,E2 -17728.51} C_VEL
LIN {X 0,Y 270.421,Z 676.872,A -85,B 0,C 180,E1 -17730,E2 -17730} C_VEL
LIN {X 0,Y 269.754,Z 676.579,A -85,B 0,C 180,E1 -17732.987,E2 -17732.987} C_VEL
LIN {X 0,Y 269.523,Z 675.821,A -85,B 0,C 180,E1 -17734.487,E2 -17734.487} C_VEL
LIN {X 0,Y 269.096,Z 672.969,A -85,B 0,C 180,E1 -17737.504,E2 -17737.504} C_VEL
LIN {X 0,Y 269.086,Z 668.454,A -85,B 0,C 180,E1 -17740.535,E2 -17740.535} C_VEL
LIN {X 0,Y 269.601,Z 663.869,A -85,B 0,C 180,E1 -17742.802,E2 -17742.802} C_VEL
LIN {X 0,Y 270.783,Z 657.082,A -85,B 0,C 180,E1 -17745.429,E2 -17745.429} C_VEL
LIN {X 0,Y 271.612,Z 652.469,A -85,B 0,C 180,E1 -17746.924,E2 -17746.924} C_VEL
LIN {X 0,Y 273.609,Z 644.36,A -85,B 0,C 180,E1 -17749.117,E2 -17749.117} C_VEL
LIN {X 0,Y 275.601,Z 636.247,A -85,B 0,C 180,E1 -17750.917,E2 -17750.917} C_VEL
LIN {X 0,Y 277.108,Z 625.482,A -85,B 0,C 180,E1 -17752.951,E2 -17752.951} C_VEL
LIN {X 0,Y 278.495,Z 613.555,A -85,B 0,C 180,E1 -17754.832,E2 -17754.832} C_VEL
LIN {X 0,Y 278.902,Z 602.333,A -85,B 0,C 180,E1 -17756.368,E2 -17756.368} C_VEL
LIN {X 0,Y 278.25,Z 590.18,A -85,B 0,C 180,E1 -17757.868,E2 -17757.868} C_VEL
LIN {X 0,Y 276.841,Z 578.224,A -85,B 0,C 180,E1 -17759.228,E2 -17759.228} C_VEL
LIN {X 0,Y 274.304,Z 565.899,A -85,B 0,C 180,E1 -17760.574,E2 -17760.574} C_VEL
LIN {X 0,Y 272.998,Z 560.943,A -85,B 0,C 180,E1 -17761.108,E2 -17761.108} C_VEL
LIN {X 0,Y 272.18,Z 557.158,A -85,B 0,C 180,E1 -17761.477,E2 -17761.477} C_VEL
LIN {X 0,Y 274.055,Z 547.251,A -85,B 0,C 180,E1 -17766.145,E2 -17766.145} C_VEL
LIN {X 0,Y 275.272,Z 542.016,A -85,B 0,C 180,E1 -17768.72,E2 -17768.72} C_VEL
LIN {X 0,Y 274.952,Z 538.384,A -85,B 0,C 180,E1 -17770.74,E2 -17770.74} C_VEL
LIN {X 0,Y 274.027,Z 532.852,A -85,B 0,C 180,E1 -17774.101,E2 -17774.101} C_VEL
LIN {X 0,Y 272.773,Z 526.649,A -85,B 0,C 180,E1 -17778.348,E2 -17778.348} C_VEL
LIN {X 0,Y 271.657,Z 521.365,A -85,B 0,C 180,E1 -17782.559,E2 -17782.559} C_VEL
LIN {X 0,Y 270.651,Z 516.74,A -85,B 0,C 180,E1 -17786.955,E2 -17786.955} C_VEL
LIN {X 0,Y 270.202,Z 514.825,A -85,B 0,C 180,E1 -17789.131,E2 -17789.131} C_VEL
LIN {X 0,Y 270.266,Z 514.818,A -85,B 0,C 180,E1 -17792.146,E2 -17792.146} C_VEL
LIN {X 0,Y 270.28,Z 514.81,A -85,B 0,C 180,E1 -17795.519,E2 -17795.519} C_VEL
LIN {X 0,Y 270.304,Z 514.813,A -85,B 0,C 180,E1 -17800.245,E2 -17800.245} C_VEL
LIN {X 0,Y 270.406,Z 514.795,A -85,B 0,C 180,E1 -17804.936,E2 -17804.936} C_VEL
LIN {X 0,Y 270.445,Z 514.793,A -85,B 0,C 180,E1 -17809.519,E2 -17809.519} C_VEL
LIN {X 0,Y 270.615,Z 514.769,A -85,B 0,C 180,E1 -17812.539,E2 -17812.539} C_VEL
LIN {X 0,Y 270.786,Z 514.754,A -85,B 0,C 180,E1 -17818.513,E2 -17818.513} C_VEL
LIN {X 0,Y 270.79,Z 514.755,A -85,B 0,C 180,E1 -17821.488,E2 -17821.488} C_VEL
LIN {X 0,Y 270.631,Z 514.777,A -85,B 0,C 180,E1 -17822.978,E2 -17822.978} C_VEL
LIN {X 0,Y 271.297,Z 517.15,A -85,B 0,C 180,E1 -17823.342,E2 -17823.342} C_VEL
LIN {X 0,Y 275.851,Z 525.062,A -85,B 0,C 180,E1 -17825.043,E2 -17825.043} C_VEL
LIN {X 0,Y 279.326,Z 532.195,A -85,B 0,C 180,E1 -17826.544,E2 -17826.544} C_VEL
LIN {X 0,Y 282.568,Z 540.814,A -85,B 0,C 180,E1 -17828.304,E2 -17828.304} C_VEL
LIN {X 0,Y 285.208,Z 550.121,A -85,B 0,C 180,E1 -17830.292,E2 -17830.292} C_VEL
LIN {X 0,Y 285.867,Z 554.234,A -85,B 0,C 180,E1 -17831.164,E2 -17831.164} C_VEL
LIN {X 0,Y 283.704,Z 563.787,A -85,B 0,C 180,E1 -17832.883,E2 -17832.883} C_VEL
LIN {X 0,Y 281.397,Z 572.542,A -85,B 0,C 180,E1 -17834.833,E2 -17834.833} C_VEL
LIN {X 0,Y 278.968,Z 580.734,A -85,B 0,C 180,E1 -17837.169,E2 -17837.169} C_VEL
LIN {X 0,Y 277.113,Z 586.506,A -85,B 0,C 180,E1 -17839.251,E2 -17839.251} C_VEL
LIN {X 0,Y 275.25,Z 591.835,A -85,B 0,C 180,E1 -17841.73,E2 -17841.73} C_VEL
LIN {X 0,Y 273.669,Z 595.745,A -85,B 0,C 180,E1 -17844.261,E2 -17844.261} C_VEL
LIN {X 0,Y 272.811,Z 597.643,A -85,B 0,C 180,E1 -17845.973,E2 -17845.973} C_VEL
LIN {X 0,Y 271.808,Z 599.404,A -85,B 0,C 180,E1 -17848.463,E2 -17848.463} C_VEL
LIN {X 0,Y 271.052,Z 600.006,A -85,B 0,C 180,E1 -17851.237,E2 -17851.237} C_VEL
LIN {X 0,Y 270.667,Z 599.353,A -85,B 0,C 180,E1 -17853.808,E2 -17853.808} C_VEL
LIN {X 0,Y 270.581,Z 597.242,A -85,B 0,C 180,E1 -17856.684,E2 -17856.684} C_VEL
LIN {X 0,Y 270.835,Z 593.539,A -85,B 0,C 180,E1 -17859.567,E2 -17859.567} C_VEL
LIN {X 0,Y 271.5,Z 588.474,A -85,B 0,C 180,E1 -17862.302,E2 -17862.302} C_VEL
LIN {X 0,Y 272.278,Z 582.758,A -85,B 0,C 180,E1 -17864.637,E2 -17864.637} C_VEL
LIN {X 0,Y 273.312,Z 575.01,A -85,B 0,C 180,E1 -17867.127,E2 -17867.127} C_VEL
LIN {X 0,Y 274.579,Z 566.481,A -85,B 0,C 180,E1 -17869.312,E2 -17869.312} C_VEL
LIN {X 0,Y 275.88,Z 556.606,A -85,B 0,C 180,E1 -17871.343,E2 -17871.343} C_VEL
LIN {X 0,Y 277.205,Z 545.667,A -85,B 0,C 180,E1 -17873.164,E2 -17873.164} C_VEL
LIN {X 0,Y 277.538,Z 540.319,A -85,B 0,C 180,E1 -17873.931,E2 -17873.931} C_VEL
LIN {X 0,Y 274.668,Z 529.522,A -85,B 0,C 180,E1 -17875.497,E2 -17875.497} C_VEL
LIN {X 0,Y 270.968,Z 517.336,A -85,B 0,C 180,E1 -17876.998,E2 -17876.998} C_VEL
LIN {X 0,Y 270.207,Z 514.832,A -85,B 0,C 180,E1 -17877.281,E2 -17877.281} C_VEL
LIN {X 0,Y 270.277,Z 514.818,A -85,B 0,C 180,E1 -17882.092,E2 -17882.092} C_VEL
LIN {X 0,Y 270.244,Z 514.824,A -85,B 0,C 180,E1 -17885.537,E2 -17885.537} C_VEL
LIN {X 0,Y 270.266,Z 514.817,A -85,B 0,C 180,E1 -17890.241,E2 -17890.241} C_VEL
LIN {X 0,Y 270.382,Z 514.805,A -85,B 0,C 180,E1 -17894.934,E2 -17894.934} C_VEL
LIN {X 0,Y 270.415,Z 514.802,A -85,B 0,C 180,E1 -17899.518,E2 -17899.518} C_VEL
LIN {X 0,Y 270.568,Z 514.78,A -85,B 0,C 180,E1 -17902.537,E2 -17902.537} C_VEL
LIN {X 0,Y 270.788,Z 514.752,A -85,B 0,C 180,E1 -17908.513,E2 -17908.513} C_VEL
LIN {X 0,Y 270.789,Z 514.755,A -85,B 0,C 180,E1 -17911.487,E2 -17911.487} C_VEL
LIN {X 0,Y 270.567,Z 514.781,A -85,B 0,C 180,E1 -17917.462,E2 -17917.462} C_VEL
LIN {X 0,Y 270.414,Z 514.798,A -85,B 0,C 180,E1 -17920.482,E2 -17920.482} C_VEL
LIN {X 0,Y 270.382,Z 514.806,A -85,B 0,C 180,E1 -17925.066,E2 -17925.066} C_VEL
LIN {X 0,Y 270.301,Z 514.813,A -85,B 0,C 180,E1 -17929.755,E2 -17929.755} C_VEL
LIN {X 0,Y 270.234,Z 514.821,A -85,B 0,C 180,E1 -17934.589,E2 -17934.589} C_VEL
LIN {X 0,Y 270.212,Z 514.823,A -85,B 0,C 180,E1 -17937.915,E2 -17937.915} C_VEL
LIN {X 0,Y 270.177,Z 514.831,A -85,B 0,C 180,E1 -17941.349,E2 -17941.349} C_VEL
LIN {X 0,Y 270.202,Z 514.826,A -85,B 0,C 180,E1 -17944.905,E2 -17944.905} C_VEL
LIN {X 0,Y 270.2,Z 514.827,A -85,B 0,C 180,E1 -17948.71,E2 -17948.71} C_VEL
LIN {X 0,Y 270.159,Z 514.833,A -85,B 0,C 180,E1 -17953.247,E2 -17953.247} C_VEL
LIN {X 0,Y 270.174,Z 514.83,A -85,B 0,C 180,E1 -17957.441,E2 -17957.441} C_VEL
LIN {X 0,Y 270.209,Z 514.825,A -85,B 0,C 180,E1 -17961.374,E2 -17961.374} C_VEL
LIN {X 0,Y 270.204,Z 514.829,A -85,B 0,C 180,E1 -17965.094,E2 -17965.094} C_VEL
LIN {X 0,Y 270.203,Z 514.827,A -85,B 0,C 180,E1 -17969.13,E2 -17969.13} C_VEL
LIN {X 0,Y 270.267,Z 514.816,A -85,B 0,C 180,E1 -17972.145,E2 -17972.145} C_VEL
LIN {X 0,Y 270.24,Z 514.821,A -85,B 0,C 180,E1 -17975.537,E2 -17975.537} C_VEL
LIN {X 0,Y 270.304,Z 514.812,A -85,B 0,C 180,E1 -17980.244,E2 -17980.244} C_VEL
LIN {X 0,Y 270.405,Z 514.804,A -85,B 0,C 180,E1 -17984.935,E2 -17984.935} C_VEL
LIN {X 0,Y 270.412,Z 514.799,A -85,B 0,C 180,E1 -17989.517,E2 -17989.517} C_VEL
LIN {X 0,Y 270.568,Z 514.781,A -85,B 0,C 180,E1 -17992.537,E2 -17992.537} C_VEL
LIN {X 0,Y 270.786,Z 514.753,A -85,B 0,C 180,E1 -17998.512,E2 -17998.512} C_VEL
LIN {X 0,Y 270.784,Z 514.753,A -85,B 0,C 180,E1 -18001.487,E2 -18001.487} C_VEL
LIN {X 0,Y 270.564,Z 514.781,A -85,B 0,C 180,E1 -18007.462,E2 -18007.462} C_VEL
LIN {X 0,Y 270.414,Z 514.8,A -85,B 0,C 180,E1 -18010.482,E2 -18010.482} C_VEL
LIN {X 0,Y 270.378,Z 514.806,A -85,B 0,C 180,E1 -18015.066,E2 -18015.066} C_VEL
LIN {X 0,Y 270.262,Z 514.817,A -85,B 0,C 180,E1 -18019.758,E2 -18019.758} C_VEL
LIN {X 0,Y 270.227,Z 514.824,A -85,B 0,C 180,E1 -18024.59,E2 -18024.59} C_VEL
LIN {X 0,Y 270.201,Z 514.825,A -85,B 0,C 180,E1 -18026.108,E2 -18026.108} C_VEL
LIN {X 0,Y 269.577,Z 514.909,A -85,B 0,C 180,E1 -18027.352,E2 -18027.352} C_VEL
LIN {X 0,Y 266.726,Z 515.269,A -85,B 0,C 180,E1 -18029.379,E2 -18029.379} C_VEL
LIN {X 0,Y 264.269,Z 515.572,A -85,B 0,C 180,E1 -18031.027,E2 -18031.027} C_VEL
LIN {X 0,Y 263.201,Z 515.701,A -85,B 0,C 180,E1 -18032.305,E2 -18032.305} C_VEL
LIN {X 0,Y 263.109,Z 515.708,A -85,B 0,C 180,E1 -18032.739,E2 -18032.739} C_VEL
LIN {X 0,Y 263.183,Z 515.703,A -85,B 0,C 180,E1 -18036.763,E2 -18036.763} C_VEL
LIN {X 0,Y 263.199,Z 515.796,A -85,B 0,C 180,E1 -18038.854,E2 -18038.854} C_VEL
LIN {X 0,Y 264.496,Z 522.466,A -85,B 0,C 180,E1 -18042.653,E2 -18042.653} C_VEL
LIN {X 0,Y 266.061,Z 530.593,A -85,B 0,C 180,E1 -18047.035,E2 -18047.035} C_VEL
LIN {X 0,Y 267.498,Z 538.181,A -85,B 0,C 180,E1 -18050.909,E2 -18050.909} C_VEL
LIN {X 0,Y 267.449,Z 540.496,A -85,B 0,C 180,E1 -18052.03,E2 -18052.03} C_VEL
LIN {X 0,Y 265.758,Z 549.577,A -85,B 0,C 180,E1 -18056.265,E2 -18056.265} C_VEL
LIN {X 0,Y 264.246,Z 558.81,A -85,B 0,C 180,E1 -18060.526,E2 -18060.526} C_VEL
LIN {X 0,Y 263.134,Z 567.985,A -85,B 0,C 180,E1 -18064.701,E2 -18064.701} C_VEL
LIN {X 0,Y 264.537,Z 583.464,A -85,B 0,C 180,E1 -18065.625,E2 -18065.625} C_VEL
LIN {X 0,Y 265.423,Z 596.269,A -85,B 0,C 180,E1 -18066.689,E2 -18066.689} C_VEL
LIN {X 0,Y 265.958,Z 608.374,A -85,B 0,C 180,E1 -18067.975,E2 -18067.975} C_VEL
LIN {X 0,Y 266.097,Z 620.093,A -85,B 0,C 180,E1 -18069.516,E2 -18069.516} C_VEL
LIN {X 0,Y 265.959,Z 631.122,A -85,B 0,C 180,E1 -18071.313,E2 -18071.313} C_VEL
LIN {X 0,Y 264.725,Z 639.849,A -85,B 0,C 180,E1 -18073.02,E2 -18073.02} C_VEL
LIN {X 0,Y 263.351,Z 649.356,A -85,B 0,C 180,E1 -18075.314,E2 -18075.314} C_VEL
LIN {X 0,Y 262.614,Z 656.971,A -85,B 0,C 180,E1 -18077.638,E2 -18077.638} C_VEL
LIN {X 0,Y 262.291,Z 663.086,A -85,B 0,C 180,E1 -18079.97,E2 -18079.97} C_VEL
LIN {X 0,Y 262.34,Z 668.078,A -85,B 0,C 180,E1 -18082.4,E2 -18082.4} C_VEL
LIN {X 0,Y 262.597,Z 671.519,A -85,B 0,C 180,E1 -18084.625,E2 -18084.625} C_VEL
LIN {X 0,Y 262.862,Z 674.016,A -85,B 0,C 180,E1 -18086.935,E2 -18086.935} C_VEL
LIN {X 0,Y 263.168,Z 675.134,A -85,B 0,C 180,E1 -18088.47,E2 -18088.47} C_VEL
LIN {X 0,Y 263.398,Z 675.774,A -85,B 0,C 180,E1 -18090,E2 -18090} C_VEL
LIN {X 0,Y 262.696,Z 675.538,A -85,B 0,C 180,E1 -18093.067,E2 -18093.067} C_VEL
LIN {X 0,Y 262.442,Z 674.812,A -85,B 0,C 180,E1 -18094.608,E2 -18094.608} C_VEL
LIN {X 0,Y 262.084,Z 672.67,A -85,B 0,C 180,E1 -18097.167,E2 -18097.167} C_VEL
LIN {X 0,Y 261.961,Z 668.897,A -85,B 0,C 180,E1 -18100.043,E2 -18100.043} C_VEL
LIN {X 0,Y 262.616,Z 663.133,A -85,B 0,C 180,E1 -18103.149,E2 -18103.149} C_VEL
LIN {X 0,Y 263.857,Z 656.202,A -85,B 0,C 180,E1 -18105.959,E2 -18105.959} C_VEL
LIN {X 0,Y 265.17,Z 650.767,A -85,B 0,C 180,E1 -18107.746,E2 -18107.746} C_VEL
LIN {X 0,Y 267.303,Z 642.502,A -85,B 0,C 180,E1 -18109.987,E2 -18109.987} C_VEL
LIN {X 0,Y 268.883,Z 636.033,A -85,B 0,C 180,E1 -18111.465,E2 -18111.465} C_VEL
LIN {X 0,Y 270.535,Z 625.636,A -85,B 0,C 180,E1 -18113.542,E2 -18113.542} C_VEL
LIN {X 0,Y 272,Z 614.224,A -85,B 0,C 180,E1 -18115.428,E2 -18115.428} C_VEL
LIN {X 0,Y 272.542,Z 603.131,A -85,B 0,C 180,E1 -18117.033,E2 -18117.033} C_VEL
LIN {X 0,Y 272.072,Z 590.443,A -85,B 0,C 180,E1 -18118.718,E2 -18118.718} C_VEL
LIN {X 0,Y 270.689,Z 578.343,A -85,B 0,C 180,E1 -18120.184,E2 -18120.184} C_VEL
LIN {X 0,Y 267.962,Z 564.753,A -85,B 0,C 180,E1 -18121.782,E2 -18121.782} C_VEL
LIN {X 0,Y 266.521,Z 559.577,A -85,B 0,C 180,E1 -18122.408,E2 -18122.408} C_VEL
LIN {X 0,Y 265.612,Z 555.544,A -85,B 0,C 180,E1 -18122.85,E2 -18122.85} C_VEL
LIN {X 0,Y 267.105,Z 548.474,A -85,B 0,C 180,E1 -18126.301,E2 -18126.301} C_VEL
LIN {X 0,Y 268.364,Z 543.262,A -85,B 0,C 180,E1 -18128.941,E2 -18128.941} C_VEL
LIN {X 0,Y 268.007,Z 539.753,A -85,B 0,C 180,E1 -18130.964,E2 -18130.964} C_VEL
LIN {X 0,Y 267.003,Z 533.82,A -85,B 0,C 180,E1 -18134.709,E2 -18134.709} C_VEL
LIN {X 0,Y 265.884,Z 528.318,A -85,B 0,C 180,E1 -18138.638,E2 -18138.638} C_VEL
LIN {X 0,Y 264.859,Z 523.299,A -85,B 0,C 180,E1 -18142.755,E2 -18142.755} C_VEL
LIN {X 0,Y 264.145,Z 519.852,A -85,B 0,C 180,E1 -18146.032,E2 -18146.032} C_VEL
LIN {X 0,Y 263.155,Z 515.697,A -85,B 0,C 180,E1 -18150.885,E2 -18150.885} C_VEL
LIN {X 0,Y 263.229,Z 515.69,A -85,B 0,C 180,E1 -18155.201,E2 -18155.201} C_VEL
LIN {X 0,Y 263.266,Z 515.684,A -85,B 0,C 180,E1 -18159.694,E2 -18159.694} C_VEL
LIN {X 0,Y 263.354,Z 515.676,A -85,B 0,C 180,E1 -18164.523,E2 -18164.523} C_VEL
LIN {X 0,Y 263.377,Z 515.671,A -85,B 0,C 180,E1 -18169.235,E2 -18169.235} C_VEL
LIN {X 0,Y 263.576,Z 515.645,A -85,B 0,C 180,E1 -18172.339,E2 -18172.339} C_VEL
LIN {X 0,Y 263.75,Z 515.63,A -85,B 0,C 180,E1 -18178.473,E2 -18178.473} C_VEL
LIN {X 0,Y 263.745,Z 515.633,A -85,B 0,C 180,E1 -18181.48,E2 -18181.48} C_VEL
LIN {X 0,Y 264.703,Z 518.542,A -85,B 0,C 180,E1 -18181.997,E2 -18181.997} C_VEL
LIN {X 0,Y 268.146,Z 524.436,A -85,B 0,C 180,E1 -18183.38,E2 -18183.38} C_VEL
LIN {X 0,Y 272.947,Z 533.672,A -85,B 0,C 180,E1 -18185.504,E2 -18185.504} C_VEL
LIN {X 0,Y 276.561,Z 543.479,A -85,B 0,C 180,E1 -18187.658,E2 -18187.658} C_VEL
LIN {X 0,Y 279.131,Z 552.906,A -85,B 0,C 180,E1 -18189.785,E2 -18189.785} C_VEL
LIN {X 0,Y 279.713,Z 556.152,A -85,B 0,C 180,E1 -18190.539,E2 -18190.539} C_VEL
LIN {X 0,Y 277.268,Z 566.274,A -85,B 0,C 180,E1 -18192.443,E2 -18192.443} C_VEL
LIN {X 0,Y 275.006,Z 574.277,A -85,B 0,C 180,E1 -18194.314,E2 -18194.314} C_VEL
LIN {X 0,Y 272.692,Z 581.661,A -85,B 0,C 180,E1 -18196.47,E2 -18196.47} C_VEL
LIN {X 0,Y 270.396,Z 588.334,A -85,B 0,C 180,E1 -18198.96,E2 -18198.96} C_VEL
LIN {X 0,Y 268.412,Z 593.44,A -85,B 0,C 180,E1 -18201.505,E2 -18201.505} C_VEL
LIN {X 0,Y 266.767,Z 597.205,A -85,B 0,C 180,E1 -18204.102,E2 -18204.102} C_VEL
LIN {X 0,Y 265.457,Z 599.706,A -85,B 0,C 180,E1 -18206.749,E2 -18206.749} C_VEL
LIN {X 0,Y 264.694,Z 600.761,A -85,B 0,C 180,E1 -18208.812,E2 -18208.812} C_VEL
LIN {X 0,Y 263.967,Z 601.059,A -85,B 0,C 180,E1 -18211.571,E2 -18211.571} C_VEL
LIN {X 0,Y 263.618,Z 600.111,A -85,B 0,C 180,E1 -18214.263,E2 -18214.263} C_VEL
LIN {X 0,Y 263.544,Z 598.003,A -85,B 0,C 180,E1 -18216.867,E2 -18216.867} C_VEL
LIN {X 0,Y 263.821,Z 594.267,A -85,B 0,C 180,E1 -18219.744,E2 -18219.744} C_VEL
LIN {X 0,Y 264.564,Z 588.767,A -85,B 0,C 180,E1 -18222.686,E2 -18222.686} C_VEL
LIN {X 0,Y 265.306,Z 583.373,A -85,B 0,C 180,E1 -18224.889,E2 -18224.889} C_VEL
LIN {X 0,Y 266.32,Z 576.019,A -85,B 0,C 180,E1 -18227.295,E2 -18227.295} C_VEL
LIN {X 0,Y 267.663,Z 567.226,A -85,B 0,C 180,E1 -18229.593,E2 -18229.593} C_VEL
LIN {X 0,Y 268.958,Z 557.578,A -85,B 0,C 180,E1 -18231.621,E2 -18231.621} C_VEL
LIN {X 0,Y 270.24,Z 547.234,A -85,B 0,C 180,E1 -18233.392,E2 -18233.392} C_VEL
LIN {X 0,Y 270.712,Z 542.006,A -85,B 0,C 180,E1 -18234.167,E2 -18234.167} C_VEL
LIN {X 0,Y 267.981,Z 531.698,A -85,B 0,C 180,E1 -18235.731,E2 -18235.731} C_VEL
LIN {X 0,Y 264.527,Z 520.138,A -85,B 0,C 180,E1 -18237.226,E2 -18237.226} C_VEL
LIN {X 0,Y 263.161,Z 515.709,A -85,B 0,C 180,E1 -18237.751,E2 -18237.751} C_VEL
LIN {X 0,Y 263.207,Z 515.701,A -85,B 0,C 180,E1 -18241.783,E2 -18241.783} C_VEL
LIN {X 0,Y 263.206,Z 515.701,A -85,B 0,C 180,E1 -18245.212,E2 -18245.212} C_VEL
LIN {X 0,Y 263.243,Z 515.695,A -85,B 0,C 180,E1 -18249.691,E2 -18249.691} C_VEL
LIN {X 0,Y 263.328,Z 515.682,A -85,B 0,C 180,E1 -18254.52,E2 -18254.52} C_VEL
LIN {X 0,Y 263.357,Z 515.682,A -85,B 0,C 180,E1 -18259.233,E2 -18259.233} C_VEL
LIN {X 0,Y 263.531,Z 515.656,A -85,B 0,C 180,E1 -18262.337,E2 -18262.337} C_VEL
LIN {X 0,Y 263.753,Z 515.628,A -85,B 0,C 180,E1 -18268.473,E2 -18268.473} C_VEL
LIN {X 0,Y 263.753,Z 515.631,A -85,B 0,C 180,E1 -18271.527,E2 -18271.527} C_VEL
LIN {X 0,Y 263.531,Z 515.656,A -85,B 0,C 180,E1 -18277.663,E2 -18277.663} C_VEL
LIN {X 0,Y 263.354,Z 515.678,A -85,B 0,C 180,E1 -18280.766,E2 -18280.766} C_VEL
LIN {X 0,Y 263.328,Z 515.683,A -85,B 0,C 180,E1 -18285.479,E2 -18285.479} C_VEL
LIN {X 0,Y 263.266,Z 515.689,A -85,B 0,C 180,E1 -18290.306,E2 -18290.306} C_VEL
LIN {X 0,Y 263.181,Z 515.701,A -85,B 0,C 180,E1 -18295.294,E2 -18295.294} C_VEL
LIN {X 0,Y 263.142,Z 515.706,A -85,B 0,C 180,E1 -18298.734,E2 -18298.734} C_VEL
LIN {X 0,Y 263.131,Z 515.705,A -85,B 0,C 180,E1 -18302.288,E2 -18302.288} C_VEL
LIN {X 0,Y 263.182,Z 515.701,A -85,B 0,C 180,E1 -18306.762,E2 -18306.762} C_VEL
LIN {X 0,Y 263.094,Z 515.71,A -85,B 0,C 180,E1 -18309.875,E2 -18309.875} C_VEL
LIN {X 0,Y 263.104,Z 515.708,A -85,B 0,C 180,E1 -18313.988,E2 -18313.988} C_VEL
LIN {X 0,Y 263.127,Z 515.707,A -85,B 0,C 180,E1 -18318.406,E2 -18318.406} C_VEL
LIN {X 0,Y 263.184,Z 515.702,A -85,B 0,C 180,E1 -18323.237,E2 -18323.237} C_VEL
LIN {X 0,Y 263.136,Z 515.705,A -85,B 0,C 180,E1 -18327.711,E2 -18327.711} C_VEL
LIN {X 0,Y 263.204,Z 515.696,A -85,B 0,C 180,E1 -18331.783,E2 -18331.783} C_VEL
LIN {X 0,Y 263.203,Z 515.7,A -85,B 0,C 180,E1 -18335.212,E2 -18335.212} C_VEL
LIN {X 0,Y 263.265,Z 515.688,A -85,B 0,C 180,E1 -18339.693,E2 -18339.693} C_VEL
LIN {X 0,Y 263.353,Z 515.679,A -85,B 0,C 180,E1 -18344.522,E2 -18344.522} C_VEL
LIN {X 0,Y 263.355,Z 515.68,A -85,B 0,C 180,E1 -18349.233,E2 -18349.233} C_VEL
LIN {X 0,Y 263.531,Z 515.657,A -85,B 0,C 180,E1 -18352.337,E2 -18352.337} C_VEL
LIN {X 0,Y 263.75,Z 515.63,A -85,B 0,C 180,E1 -18358.473,E2 -18358.473} C_VEL
LIN {X 0,Y 263.748,Z 515.629,A -85,B 0,C 180,E1 -18361.527,E2 -18361.527} C_VEL
LIN {X 0,Y 263.528,Z 515.656,A -85,B 0,C 180,E1 -18367.663,E2 -18367.663} C_VEL
LIN {X 0,Y 263.356,Z 515.681,A -85,B 0,C 180,E1 -18370.766,E2 -18370.766} C_VEL
LIN {X 0,Y 263.325,Z 515.682,A -85,B 0,C 180,E1 -18375.479,E2 -18375.479} C_VEL
LIN {X 0,Y 263.239,Z 515.693,A -85,B 0,C 180,E1 -18380.308,E2 -18380.308} C_VEL
LIN {X 0,Y 263.17,Z 515.702,A -85,B 0,C 180,E1 -18385.295,E2 -18385.295} C_VEL
LIN {X 0,Y 263.136,Z 515.709,A -85,B 0,C 180,E1 -18388.734,E2 -18388.734} C_VEL
LIN {X 0,Y 263.109,Z 515.708,A -85,B 0,C 180,E1 -18392.739,E2 -18392.739} C_VEL
LIN {X 0,Y 262.445,Z 515.792,A -85,B 0,C 180,E1 -18393.59,E2 -18393.59} C_VEL
LIN {X 0,Y 259.684,Z 516.139,A -85,B 0,C 180,E1 -18394.929,E2 -18394.929} C_VEL
LIN {X 0,Y 256.857,Z 516.492,A -85,B 0,C 180,E1 -18396.295,E2 -18396.295} C_VEL
LIN {X 0,Y 256.126,Z 516.581,A -85,B 0,C 180,E1 -18397.177,E2 -18397.177} C_VEL
LIN {X 0,Y 256.179,Z 516.747,A -85,B 0,C 180,E1 -18398.493,E2 -18398.493} C_VEL
LIN {X 0,Y 257.649,Z 524.467,A -85,B 0,C 180,E1 -18402.995,E2 -18402.995} C_VEL
LIN {X 0,Y 259.156,Z 532.333,A -85,B 0,C 180,E1 -18407.315,E2 -18407.315} C_VEL
LIN {X 0,Y 260.398,Z 538.613,A -85,B 0,C 180,E1 -18410.624,E2 -18410.624} C_VEL
LIN {X 0,Y 260.453,Z 540.622,A -85,B 0,C 180,E1 -18411.638,E2 -18411.638} C_VEL
LIN {X 0,Y 259.019,Z 548.186,A -85,B 0,C 180,E1 -18415.264,E2 -18415.264} C_VEL
LIN {X 0,Y 257.415,Z 557.395,A -85,B 0,C 180,E1 -18419.663,E2 -18419.663} C_VEL
LIN {X 0,Y 256.14,Z 567,A -85,B 0,C 180,E1 -18424.192,E2 -18424.192} C_VEL
LIN {X 0,Y 257.521,Z 582.642,A -85,B 0,C 180,E1 -18425.163,E2 -18425.163} C_VEL
LIN {X 0,Y 258.358,Z 595.434,A -85,B 0,C 180,E1 -18426.264,E2 -18426.264} C_VEL
LIN {X 0,Y 258.931,Z 608.169,A -85,B 0,C 180,E1 -18427.667,E2 -18427.667} C_VEL
LIN {X 0,Y 259,Z 618.997,A -85,B 0,C 180,E1 -18429.136,E2 -18429.136} C_VEL
LIN {X 0,Y 258.924,Z 630.092,A -85,B 0,C 180,E1 -18430.991,E2 -18430.991} C_VEL
LIN {X 0,Y 257.53,Z 640.512,A -85,B 0,C 180,E1 -18433.123,E2 -18433.123} C_VEL
LIN {X 0,Y 256.262,Z 649.019,A -85,B 0,C 180,E1 -18435.305,E2 -18435.305} C_VEL
LIN {X 0,Y 255.545,Z 656.506,A -85,B 0,C 180,E1 -18437.694,E2 -18437.694} C_VEL
LIN {X 0,Y 255.217,Z 663.394,A -85,B 0,C 180,E1 -18440.49,E2 -18440.49} C_VEL
LIN {X 0,Y 255.315,Z 667.742,A -85,B 0,C 180,E1 -18442.794,E2 -18442.794} C_VEL
LIN {X 0,Y 255.661,Z 671.218,A -85,B 0,C 180,E1 -18445.27,E2 -18445.27} C_VEL
LIN {X 0,Y 255.824,Z 672.793,A -85,B 0,C 180,E1 -18446.851,E2 -18446.851} C_VEL
LIN {X 0,Y 256.143,Z 673.949,A -85,B 0,C 180,E1 -18448.428,E2 -18448.428} C_VEL
LIN {X 0,Y 256.374,Z 674.651,A -85,B 0,C 180,E1 -18450,E2 -18450} C_VEL
LIN {X 0,Y 255.905,Z 674.774,A -85,B 0,C 180,E1 -18451.574,E2 -18451.574} C_VEL
LIN {X 0,Y 255.636,Z 674.497,A -85,B 0,C 180,E1 -18453.152,E2 -18453.152} C_VEL
LIN {X 0,Y 255.365,Z 673.801,A -85,B 0,C 180,E1 -18454.736,E2 -18454.736} C_VEL
LIN {X 0,Y 255.029,Z 671.872,A -85,B 0,C 180,E1 -18457.218,E2 -18457.218} C_VEL
LIN {X 0,Y 254.89,Z 668.077,A -85,B 0,C 180,E1 -18460.325,E2 -18460.325} C_VEL
LIN {X 0,Y 255.344,Z 664.02,A -85,B 0,C 180,E1 -18462.72,E2 -18462.72} C_VEL
LIN {X 0,Y 256.291,Z 658.92,A -85,B 0,C 180,E1 -18465.101,E2 -18465.101} C_VEL
LIN {X 0,Y 257.663,Z 652.656,A -85,B 0,C 180,E1 -18467.46,E2 -18467.46} C_VEL
LIN {X 0,Y 259.772,Z 645.095,A -85,B 0,C 180,E1 -18469.766,E2 -18469.766} C_VEL
LIN {X 0,Y 261.891,Z 637.596,A -85,B 0,C 180,E1 -18471.654,E2 -18471.654} C_VEL
LIN {X 0,Y 263.826,Z 626.746,A -85,B 0,C 180,E1 -18473.969,E2 -18473.969} C_VEL
LIN {X 0,Y 265.56,Z 614.942,A -85,B 0,C 180,E1 -18476.051,E2 -18476.051} C_VEL
LIN {X 0,Y 266.267,Z 604.128,A -85,B 0,C 180,E1 -18477.724,E2 -18477.724} C_VEL
LIN {X 0,Y 265.92,Z 591.124,A -85,B 0,C 180,E1 -18479.548,E2 -18479.548} C_VEL
LIN {X 0,Y 264.499,Z 577.944,A -85,B 0,C 180,E1 -18481.279,E2 -18481.279} C_VEL
LIN {X 0,Y 261.815,Z 564.157,A -85,B 0,C 180,E1 -18483.013,E2 -18483.013} C_VEL
LIN {X 0,Y 259.99,Z 557.812,A -85,B 0,C 180,E1 -18483.866,E2 -18483.866} C_VEL
LIN {X 0,Y 259.197,Z 553.866,A -85,B 0,C 180,E1 -18484.349,E2 -18484.349} C_VEL
LIN {X 0,Y 261.249,Z 545.349,A -85,B 0,C 180,E1 -18488.726,E2 -18488.726} C_VEL
LIN {X 0,Y 261.338,Z 542.768,A -85,B 0,C 180,E1 -18490.197,E2 -18490.197} C_VEL
LIN {X 0,Y 260.335,Z 536.704,A -85,B 0,C 180,E1 -18494.049,E2 -18494.049} C_VEL
LIN {X 0,Y 259.17,Z 530.72,A -85,B 0,C 180,E1 -18498.366,E2 -18498.366} C_VEL
LIN {X 0,Y 258.248,Z 526.171,A -85,B 0,C 180,E1 -18502.112,E2 -18502.112} C_VEL
LIN {X 0,Y 257.574,Z 523.069,A -85,B 0,C 180,E1 -18505.041,E2 -18505.041} C_VEL
LIN {X 0,Y 256.801,Z 519.754,A -85,B 0,C 180,E1 -18508.669,E2 -18508.669} C_VEL
LIN {X 0,Y 256.172,Z 516.566,A -85,B 0,C 180,E1 -18512.92,E2 -18512.92} C_VEL
LIN {X 0,Y 256.17,Z 516.566,A -85,B 0,C 180,E1 -18515.7,E2 -18515.7} C_VEL
LIN {X 0,Y 256.169,Z 516.566,A -85,B 0,C 180,E1 -18519.105,E2 -18519.105} C_VEL
LIN {X 0,Y 256.303,Z 516.558,A -85,B 0,C 180,E1 -18524.086,E2 -18524.086} C_VEL
LIN {X 0,Y 256.313,Z 516.549,A -85,B 0,C 180,E1 -18528.934,E2 -18528.934} C_VEL
LIN {X 0,Y 256.544,Z 516.52,A -85,B 0,C 180,E1 -18532.128,E2 -18532.128} C_VEL
LIN {X 0,Y 256.713,Z 516.506,A -85,B 0,C 180,E1 -18538.432,E2 -18538.432} C_VEL
LIN {X 0,Y 256.751,Z 516.502,A -85,B 0,C 180,E1 -18539.804,E2 -18539.804} C_VEL
LIN {X 0,Y 257.674,Z 519.248,A -85,B 0,C 180,E1 -18540.323,E2 -18540.323} C_VEL
LIN {X 0,Y 259.046,Z 520.938,A -85,B 0,C 180,E1 -18540.855,E2 -18540.855} C_VEL
LIN {X 0,Y 264.575,Z 531.436,A -85,B 0,C 180,E1 -18543.426,E2 -18543.426} C_VEL
LIN {X 0,Y 268.234,Z 539.305,A -85,B 0,C 180,E1 -18545.348,E2 -18545.348} C_VEL
LIN {X 0,Y 271.201,Z 548.218,A -85,B 0,C 180,E1 -18547.445,E2 -18547.445} C_VEL
LIN {X 0,Y 273.332,Z 557.194,A -85,B 0,C 180,E1 -18549.621,E2 -18549.621} C_VEL
LIN {X 0,Y 273.564,Z 558.69,A -85,B 0,C 180,E1 -18549.987,E2 -18549.987} C_VEL
LIN {X 0,Y 271.289,Z 567.344,A -85,B 0,C 180,E1 -18551.668,E2 -18551.668} C_VEL
LIN {X 0,Y 268.484,Z 576.499,A -85,B 0,C 180,E1 -18553.896,E2 -18553.896} C_VEL
LIN {X 0,Y 266.064,Z 583.679,A -85,B 0,C 180,E1 -18556.103,E2 -18556.103} C_VEL
LIN {X 0,Y 263.661,Z 590.145,A -85,B 0,C 180,E1 -18558.655,E2 -18558.655} C_VEL
LIN {X 0,Y 261.576,Z 595.09,A -85,B 0,C 180,E1 -18561.268,E2 -18561.268} C_VEL
LIN {X 0,Y 259.861,Z 598.692,A -85,B 0,C 180,E1 -18563.934,E2 -18563.934} C_VEL
LIN {X 0,Y 258.65,Z 600.764,A -85,B 0,C 180,E1 -18566.275,E2 -18566.275} C_VEL
LIN {X 0,Y 257.483,Z 602.107,A -85,B 0,C 180,E1 -18569.427,E2 -18569.427} C_VEL
LIN {X 0,Y 256.88,Z 602.016,A -85,B 0,C 180,E1 -18571.99,E2 -18571.99} C_VEL
LIN {X 0,Y 256.544,Z 600.485,A -85,B 0,C 180,E1 -18575.121,E2 -18575.121} C_VEL
LIN {X 0,Y 256.577,Z 597.479,A -85,B 0,C 180,E1 -18578.142,E2 -18578.142} C_VEL
LIN {X 0,Y 257.033,Z 593.146,A -85,B 0,C 180,E1 -18581.014,E2 -18581.014} C_VEL
LIN {X 0,Y 257.768,Z 588.109,A -85,B 0,C 180,E1 -18583.492,E2 -18583.492} C_VEL
LIN {X 0,Y 258.721,Z 581.467,A -85,B 0,C 180,E1 -18586.044,E2 -18586.044} C_VEL
LIN {X 0,Y 259.717,Z 574.639,A -85,B 0,C 180,E1 -18588.16,E2 -18588.16} C_VEL
LIN {X 0,Y 261.031,Z 565.956,A -85,B 0,C 180,E1 -18590.356,E2 -18590.356} C_VEL
LIN {X 0,Y 262.351,Z 556.425,A -85,B 0,C 180,E1 -18592.323,E2 -18592.323} C_VEL
LIN {X 0,Y 263.672,Z 545.769,A -85,B 0,C 180,E1 -18594.098,E2 -18594.098} C_VEL
LIN {X 0,Y 263.66,Z 542.779,A -85,B 0,C 180,E1 -18594.566,E2 -18594.566} C_VEL
LIN {X 0,Y 261.153,Z 533.285,A -85,B 0,C 180,E1 -18596.054,E2 -18596.054} C_VEL
LIN {X 0,Y 257.685,Z 521.824,A -85,B 0,C 180,E1 -18597.586,E2 -18597.586} C_VEL
LIN {X 0,Y 256.11,Z 516.586,A -85,B 0,C 180,E1 -18598.239,E2 -18598.239} C_VEL
LIN {X 0,Y 256.147,Z 516.579,A -85,B 0,C 180,E1 -18602.196,E2 -18602.196} C_VEL
LIN {X 0,Y 256.147,Z 516.579,A -85,B 0,C 180,E1 -18605.697,E2 -18605.697} C_VEL
LIN {X 0,Y 256.153,Z 516.578,A -85,B 0,C 180,E1 -18609.103,E2 -18609.103} C_VEL
LIN {X 0,Y 256.263,Z 516.562,A -85,B 0,C 180,E1 -18614.082,E2 -18614.082} C_VEL
LIN {X 0,Y 256.293,Z 516.563,A -85,B 0,C 180,E1 -18617.327,E2 -18617.327} C_VEL
LIN {X 0,Y 256.438,Z 516.54,A -85,B 0,C 180,E1 -18620.622,E2 -18620.622} C_VEL
LIN {X 0,Y 256.464,Z 516.538,A -85,B 0,C 180,E1 -18623.707,E2 -18623.707} C_VEL
LIN {X 0,Y 256.716,Z 516.505,A -85,B 0,C 180,E1 -18628.431,E2 -18628.431} C_VEL
LIN {X 0,Y 256.716,Z 516.507,A -85,B 0,C 180,E1 -18631.569,E2 -18631.569} C_VEL
LIN {X 0,Y 256.462,Z 516.536,A -85,B 0,C 180,E1 -18636.293,E2 -18636.293} C_VEL
LIN {X 0,Y 256.431,Z 516.542,A -85,B 0,C 180,E1 -18639.465,E2 -18639.465} C_VEL
LIN {X 0,Y 256.242,Z 516.564,A -85,B 0,C 180,E1 -18644.291,E2 -18644.291} C_VEL
LIN {X 0,Y 256.188,Z 516.571,A -85,B 0,C 180,E1 -18647.563,E2 -18647.563} C_VEL
LIN {X 0,Y 256.159,Z 516.578,A -85,B 0,C 180,E1 -18651.118,E2 -18651.118} C_VEL
LIN {X 0,Y 256.166,Z 516.576,A -85,B 0,C 180,E1 -18655.126,E2 -18655.126} C_VEL
LIN {X 0,Y 256.061,Z 516.588,A -85,B 0,C 180,E1 -18659.606,E2 -18659.606} C_VEL
LIN {X 0,Y 256.069,Z 516.587,A -85,B 0,C 180,E1 -18663.293,E2 -18663.293} C_VEL
LIN {X 0,Y 256.115,Z 516.583,A -85,B 0,C 180,E1 -18667.27,E2 -18667.27} C_VEL
LIN {X 0,Y 256.062,Z 516.585,A -85,B 0,C 180,E1 -18672.178,E2 -18672.178} C_VEL
LIN {X 0,Y 256.051,Z 516.589,A -85,B 0,C 180,E1 -18676.67,E2 -18676.67} C_VEL
LIN {X 0,Y 256.074,Z 516.587,A -85,B 0,C 180,E1 -18680.858,E2 -18680.858} C_VEL
LIN {X 0,Y 256.132,Z 516.579,A -85,B 0,C 180,E1 -18682.867,E2 -18682.867} C_VEL
LIN {X 0,Y 256.07,Z 516.587,A -85,B 0,C 180,E1 -18686.707,E2 -18686.707} C_VEL
LIN {X 0,Y 256.116,Z 516.578,A -85,B 0,C 180,E1 -18690.4,E2 -18690.4} C_VEL
LIN {X 0,Y 256.173,Z 516.576,A -85,B 0,C 180,E1 -18694.869,E2 -18694.869} C_VEL
LIN {X 0,Y 256.165,Z 516.576,A -85,B 0,C 180,E1 -18699.104,E2 -18699.104} C_VEL
LIN {X 0,Y 256.302,Z 516.556,A -85,B 0,C 180,E1 -18704.085,E2 -18704.085} C_VEL
LIN {X 0,Y 256.298,Z 516.56,A -85,B 0,C 180,E1 -18708.933,E2 -18708.933} C_VEL
LIN {X 0,Y 256.494,Z 516.533,A -85,B 0,C 180,E1 -18712.125,E2 -18712.125} C_VEL
LIN {X 0,Y 256.494,Z 516.534,A -85,B 0,C 180,E1 -18716.858,E2 -18716.858} C_VEL
LIN {X 0,Y 256.752,Z 516.5,A -85,B 0,C 180,E1 -18720,E2 -18720} C_VEL
LIN {X 0,Y 256.482,Z 516.535,A -85,B 0,C 180,E1 -18723.141,E2 -18723.141} C_VEL
LIN {X 0,Y 256.47,Z 516.535,A -85,B 0,C 180,E1 -18727.875,E2 -18727.875} C_VEL
LIN {X 0,Y 256.298,Z 516.559,A -85,B 0,C 180,E1 -18731.066,E2 -18731.066} C_VEL
LIN {X 0,Y 256.239,Z 516.564,A -85,B 0,C 180,E1 -18734.291,E2 -18734.291} C_VEL
LIN {X 0,Y 256.178,Z 516.572,A -85,B 0,C 180,E1 -18737.564,E2 -18737.564} C_VEL
LIN {X 0,Y 256.143,Z 516.577,A -85,B 0,C 180,E1 -18741.11,E2 -18741.11} C_VEL
LIN {X 0,Y 256.135,Z 516.58,A -85,B 0,C 180,E1 -18745.112,E2 -18745.112} C_VEL
LIN {X 0,Y 256.056,Z 516.587,A -85,B 0,C 180,E1 -18749.607,E2 -18749.607} C_VEL
LIN {X 0,Y 256.066,Z 516.588,A -85,B 0,C 180,E1 -18753.293,E2 -18753.293} C_VEL
LIN {X 0,Y 256.126,Z 516.581,A -85,B 0,C 180,E1 -18757.177,E2 -18757.177} C_VEL
LIN {X 0,Y 255.788,Z 516.978,A -85,B 0,C 180,E1 -18758.051,E2 -18758.051} C_VEL
LIN {X 0,Y 255.095,Z 517.973,A -85,B 0,C 180,E1 -18758.896,E2 -18758.896} C_VEL
LIN {X 0,Y 251.446,Z 524.133,A -85,B 0,C 180,E1 -18762.142,E2 -18762.142} C_VEL
LIN {X 0,Y 250.895,Z 526.455,A -85,B 0,C 180,E1 -18763.389,E2 -18763.389} C_VEL
LIN {X 0,Y 250.954,Z 527.199,A -85,B 0,C 180,E1 -18763.81,E2 -18763.81} C_VEL
LIN {X 0,Y 252.433,Z 534.825,A -85,B 0,C 180,E1 -18768.073,E2 -18768.073} C_VEL
LIN {X 0,Y 253.398,Z 540.193,A -85,B 0,C 180,E1 -18770.948,E2 -18770.948} C_VEL
LIN {X 0,Y 252.759,Z 544.604,A -85,B 0,C 180,E1 -18773.164,E2 -18773.164} C_VEL
LIN {X 0,Y 251.247,Z 552.496,A -85,B 0,C 180,E1 -18777.053,E2 -18777.053} C_VEL
LIN {X 0,Y 249.539,Z 563.286,A -85,B 0,C 180,E1 -18782.309,E2 -18782.309} C_VEL
LIN {X 0,Y 249.166,Z 566.066,A -85,B 0,C 180,E1 -18783.667,E2 -18783.667} C_VEL
LIN {X 0,Y 250.481,Z 580.933,A -85,B 0,C 180,E1 -18784.613,E2 -18784.613} C_VEL
LIN {X 0,Y 251.333,Z 593.935,A -85,B 0,C 180,E1 -18785.751,E2 -18785.751} C_VEL
LIN {X 0,Y 251.803,Z 605.836,A -85,B 0,C 180,E1 -18787.08,E2 -18787.08} C_VEL
LIN {X 0,Y 252.01,Z 616.419,A -85,B 0,C 180,E1 -18788.529,E2 -18788.529} C_VEL
LIN {X 0,Y 251.877,Z 627.873,A -85,B 0,C 180,E1 -18790.438,E2 -18790.438} C_VEL
LIN {X 0,Y 251.629,Z 632.159,A -85,B 0,C 180,E1 -18791.265,E2 -18791.265} C_VEL
LIN {X 0,Y 250.244,Z 641.482,A -85,B 0,C 180,E1 -18793.349,E2 -18793.349} C_VEL
LIN {X 0,Y 249.05,Z 649.992,A -85,B 0,C 180,E1 -18795.705,E2 -18795.705} C_VEL
LIN {X 0,Y 248.419,Z 657.107,A -85,B 0,C 180,E1 -18798.164,E2 -18798.164} C_VEL
LIN {X 0,Y 248.163,Z 663.549,A -85,B 0,C 180,E1 -18801.039,E2 -18801.039} C_VEL
LIN {X 0,Y 248.377,Z 667.753,A -85,B 0,C 180,E1 -18803.501,E2 -18803.501} C_VEL
LIN {X 0,Y 248.626,Z 669.933,A -85,B 0,C 180,E1 -18805.136,E2 -18805.136} C_VEL
LIN {X 0,Y 248.785,Z 671.566,A -85,B 0,C 180,E1 -18806.761,E2 -18806.761} C_VEL
LIN {X 0,Y 249.116,Z 672.763,A -85,B 0,C 180,E1 -18808.384,E2 -18808.384} C_VEL
LIN {X 0,Y 249.349,Z 673.505,A -85,B 0,C 180,E1 -18810,E2 -18810} C_VEL
LIN {X 0,Y 248.865,Z 673.697,A -85,B 0,C 180,E1 -18811.618,E2 -18811.618} C_VEL
LIN {X 0,Y 248.573,Z 673.454,A -85,B 0,C 180,E1 -18813.242,E2 -18813.242} C_VEL
LIN {X 0,Y 248.291,Z 672.793,A -85,B 0,C 180,E1 -18814.871,E2 -18814.871} C_VEL
LIN {X 0,Y 247.954,Z 671.124,A -85,B 0,C 180,E1 -18817.235,E2 -18817.235} C_VEL
LIN {X 0,Y 247.832,Z 667.238,A -85,B 0,C 180,E1 -18820.622,E2 -18820.622} C_VEL
LIN {X 0,Y 248.365,Z 663.268,A -85,B 0,C 180,E1 -18823.084,E2 -18823.084} C_VEL
LIN {X 0,Y 249.383,Z 658.284,A -85,B 0,C 180,E1 -18825.529,E2 -18825.529} C_VEL
LIN {X 0,Y 250.33,Z 653.854,A -85,B 0,C 180,E1 -18827.341,E2 -18827.341} C_VEL
LIN {X 0,Y 252.68,Z 646.107,A -85,B 0,C 180,E1 -18829.921,E2 -18829.921} C_VEL
LIN {X 0,Y 254.853,Z 638.984,A -85,B 0,C 180,E1 -18831.857,E2 -18831.857} C_VEL
LIN {X 0,Y 256.919,Z 628.804,A -85,B 0,C 180,E1 -18834.226,E2 -18834.226} C_VEL
LIN {X 0,Y 258.958,Z 617.337,A -85,B 0,C 180,E1 -18836.414,E2 -18836.414} C_VEL
LIN {X 0,Y 259.926,Z 606.381,A -85,B 0,C 180,E1 -18838.241,E2 -18838.241} C_VEL
LIN {X 0,Y 259.96,Z 594.147,A -85,B 0,C 180,E1 -18840.104,E2 -18840.104} C_VEL
LIN {X 0,Y 259.159,Z 582.857,A -85,B 0,C 180,E1 -18841.698,E2 -18841.698} C_VEL
LIN {X 0,Y 257.081,Z 569.808,A -85,B 0,C 180,E1 -18843.508,E2 -18843.508} C_VEL
LIN {X 0,Y 255.137,Z 561.528,A -85,B 0,C 180,E1 -18844.668,E2 -18844.668} C_VEL
LIN {X 0,Y 253.887,Z 556.703,A -85,B 0,C 180,E1 -18845.337,E2 -18845.337} C_VEL
LIN {X 0,Y 252.918,Z 552.218,A -85,B 0,C 180,E1 -18845.952,E2 -18845.952} C_VEL
LIN {X 0,Y 254.521,Z 545.756,A -85,B 0,C 180,E1 -18849.427,E2 -18849.427} C_VEL
LIN {X 0,Y 253.817,Z 540.434,A -85,B 0,C 180,E1 -18852.798,E2 -18852.798} C_VEL
LIN {X 0,Y 252.887,Z 535.492,A -85,B 0,C 180,E1 -18856.268,E2 -18856.268} C_VEL
LIN {X 0,Y 251.949,Z 530.634,A -85,B 0,C 180,E1 -18860.091,E2 -18860.091} C_VEL
LIN {X 0,Y 251.014,Z 526.358,A -85,B 0,C 180,E1 -18863.987,E2 -18863.987} C_VEL
LIN {X 0,Y 250.273,Z 522.788,A -85,B 0,C 180,E1 -18867.755,E2 -18867.755} C_VEL
LIN {X 0,Y 249.645,Z 519.914,A -85,B 0,C 180,E1 -18871.407,E2 -18871.407} C_VEL
LIN {X 0,Y 249.129,Z 517.444,A -85,B 0,C 180,E1 -18875.412,E2 -18875.412} C_VEL
LIN {X 0,Y 249.114,Z 517.451,A -85,B 0,C 180,E1 -18880.212,E2 -18880.212} C_VEL
LIN {X 0,Y 249.245,Z 517.439,A -85,B 0,C 180,E1 -18883.622,E2 -18883.622} C_VEL
LIN {X 0,Y 249.256,Z 517.428,A -85,B 0,C 180,E1 -18888.617,E2 -18888.617} C_VEL
LIN {X 0,Y 249.488,Z 517.398,A -85,B 0,C 180,E1 -18891.903,E2 -18891.903} C_VEL
LIN {X 0,Y 249.427,Z 517.416,A -85,B 0,C 180,E1 -18896.77,E2 -18896.77} C_VEL
LIN {X 0,Y 249.563,Z 517.417,A -85,B 0,C 180,E1 -18897.832,E2 -18897.832} C_VEL
LIN {X 0,Y 250.537,Z 519.998,A -85,B 0,C 180,E1 -18898.393,E2 -18898.393} C_VEL
LIN {X 0,Y 252.775,Z 522.717,A -85,B 0,C 180,E1 -18899.357,E2 -18899.357} C_VEL
LIN {X 0,Y 254.029,Z 525.246,A -85,B 0,C 180,E1 -18900,E2 -18900} C_VEL
LIN {X 0,Y 254.948,Z 526.416,A -85,B 0,C 180,E1 -18900.395,E2 -18900.395} C_VEL
LIN {X 0,Y 260.486,Z 537.634,A -85,B 0,C 180,E1 -18903.359,E2 -18903.359} C_VEL
LIN {X 0,Y 263.684,Z 545.708,A -85,B 0,C 180,E1 -18905.441,E2 -18905.441} C_VEL
LIN {X 0,Y 266.092,Z 554.236,A -85,B 0,C 180,E1 -18907.589,E2 -18907.589} C_VEL
LIN {X 0,Y 267.248,Z 559.919,A -85,B 0,C 180,E1 -18909.079,E2 -18909.079} C_VEL
LIN {X 0,Y 267.305,Z 561.503,A -85,B 0,C 180,E1 -18909.459,E2 -18909.459} C_VEL
LIN {X 0,Y 264.394,Z 571.556,A -85,B 0,C 180,E1 -18911.567,E2 -18911.567} C_VEL
LIN {X 0,Y 261.878,Z 579.214,A -85,B 0,C 180,E1 -18913.582,E2 -18913.582} C_VEL
LIN {X 0,Y 259.48,Z 585.732,A -85,B 0,C 180,E1 -18915.715,E2 -18915.715} C_VEL
LIN {X 0,Y 256.947,Z 591.934,A -85,B 0,C 180,E1 -18918.334,E2 -18918.334} C_VEL
LIN {X 0,Y 254.751,Z 596.732,A -85,B 0,C 180,E1 -18921.017,E2 -18921.017} C_VEL
LIN {X 0,Y 253.067,Z 599.997,A -85,B 0,C 180,E1 -18923.586,E2 -18923.586} C_VEL
LIN {X 0,Y 251.502,Z 602.345,A -85,B 0,C 180,E1 -18926.592,E2 -18926.592} C_VEL
LIN {X 0,Y 250.428,Z 603.27,A -85,B 0,C 180,E1 -18929.542,E2 -18929.542} C_VEL
LIN {X 0,Y 249.782,Z 602.913,A -85,B 0,C 180,E1 -18932.424,E2 -18932.424} C_VEL
LIN {X 0,Y 249.501,Z 601.355,A -85,B 0,C 180,E1 -18935.226,E2 -18935.226} C_VEL
LIN {X 0,Y 249.542,Z 598.235,A -85,B 0,C 180,E1 -18938.288,E2 -18938.288} C_VEL
LIN {X 0,Y 250.077,Z 593.483,A -85,B 0,C 180,E1 -18941.405,E2 -18941.405} C_VEL
LIN {X 0,Y 251.037,Z 587.079,A -85,B 0,C 180,E1 -18944.42,E2 -18944.42} C_VEL
LIN {X 0,Y 251.981,Z 580.287,A -85,B 0,C 180,E1 -18946.922,E2 -18946.922} C_VEL
LIN {X 0,Y 253.33,Z 571.72,A -85,B 0,C 180,E1 -18949.417,E2 -18949.417} C_VEL
LIN {X 0,Y 254.694,Z 562.749,A -85,B 0,C 180,E1 -18951.535,E2 -18951.535} C_VEL
LIN {X 0,Y 255.983,Z 553.265,A -85,B 0,C 180,E1 -18953.376,E2 -18953.376} C_VEL
LIN {X 0,Y 256.955,Z 545.052,A -85,B 0,C 180,E1 -18954.704,E2 -18954.704} C_VEL
LIN {X 0,Y 254.187,Z 534.484,A -85,B 0,C 180,E1 -18956.428,E2 -18956.428} C_VEL
LIN {X 0,Y 251.102,Z 524.142,A -85,B 0,C 180,E1 -18957.873,E2 -18957.873} C_VEL
LIN {X 0,Y 249.066,Z 517.464,A -85,B 0,C 180,E1 -18958.709,E2 -18958.709} C_VEL
LIN {X 0,Y 249.102,Z 517.461,A -85,B 0,C 180,E1 -18961.339,E2 -18961.339} C_VEL
LIN {X 0,Y 249.14,Z 517.452,A -85,B 0,C 180,E1 -18964.967,E2 -18964.967} C_VEL
LIN {X 0,Y 249.094,Z 517.455,A -85,B 0,C 180,E1 -18968.604,E2 -18968.604} C_VEL
LIN {X 0,Y 249.2,Z 517.445,A -85,B 0,C 180,E1 -18973.619,E2 -18973.619} C_VEL
LIN {X 0,Y 249.246,Z 517.437,A -85,B 0,C 180,E1 -18978.616,E2 -18978.616} C_VEL
LIN {X 0,Y 249.44,Z 517.412,A -85,B 0,C 180,E1 -18981.901,E2 -18981.901} C_VEL
LIN {X 0,Y 249.435,Z 517.413,A -85,B 0,C 180,E1 -18986.769,E2 -18986.769} C_VEL
LIN {X 0,Y 249.678,Z 517.381,A -85,B 0,C 180,E1 -18988.387,E2 -18988.387} C_VEL
LIN {X 0,Y 249.678,Z 517.383,A -85,B 0,C 180,E1 -18991.613,E2 -18991.613} C_VEL
LIN {X 0,Y 249.433,Z 517.412,A -85,B 0,C 180,E1 -18996.471,E2 -18996.471} C_VEL
LIN {X 0,Y 249.347,Z 517.423,A -85,B 0,C 180,E1 -18999.736,E2 -18999.736} C_VEL
LIN {X 0,Y 249.187,Z 517.444,A -85,B 0,C 180,E1 -19004.704,E2 -19004.704} C_VEL
LIN {X 0,Y 249.125,Z 517.449,A -85,B 0,C 180,E1 -19008.078,E2 -19008.078} C_VEL
LIN {X 0,Y 249.088,Z 517.457,A -85,B 0,C 180,E1 -19011.518,E2 -19011.518} C_VEL
LIN {X 0,Y 249.11,Z 517.452,A -85,B 0,C 180,E1 -19015.47,E2 -19015.47} C_VEL
LIN {X 0,Y 249.045,Z 517.463,A -85,B 0,C 180,E1 -19018.975,E2 -19018.975} C_VEL
LIN {X 0,Y 249.03,Z 517.462,A -85,B 0,C 180,E1 -19022.426,E2 -19022.426} C_VEL
LIN {X 0,Y 249.031,Z 517.462,A -85,B 0,C 180,E1 -19026.345,E2 -19026.345} C_VEL
LIN {X 0,Y 248.987,Z 517.468,A -85,B 0,C 180,E1 -19030.482,E2 -19030.482} C_VEL
LIN {X 0,Y 248.996,Z 517.467,A -85,B 0,C 180,E1 -19032.788,E2 -19032.788} C_VEL
LIN {X 0,Y 249.012,Z 517.467,A -85,B 0,C 180,E1 -19037.361,E2 -19037.361} C_VEL
LIN {X 0,Y 249.028,Z 517.461,A -85,B 0,C 180,E1 -19041.619,E2 -19041.619} C_VEL
LIN {X 0,Y 249.046,Z 517.461,A -85,B 0,C 180,E1 -19045.639,E2 -19045.639} C_VEL
LIN {X 0,Y 249.054,Z 517.458,A -85,B 0,C 180,E1 -19049.473,E2 -19049.473} C_VEL
LIN {X 0,Y 249.073,Z 517.461,A -85,B 0,C 180,E1 -19053.162,E2 -19053.162} C_VEL
LIN {X 0,Y 249.064,Z 517.46,A -85,B 0,C 180,E1 -19056.73,E2 -19056.73} C_VEL
LIN {X 0,Y 249.111,Z 517.451,A -85,B 0,C 180,E1 -19060.211,E2 -19060.211} C_VEL
LIN {X 0,Y 249.244,Z 517.436,A -85,B 0,C 180,E1 -19063.621,E2 -19063.621} C_VEL
LIN {X 0,Y 249.245,Z 517.436,A -85,B 0,C 180,E1 -19068.616,E2 -19068.616} C_VEL
LIN {X 0,Y 249.438,Z 517.411,A -85,B 0,C 180,E1 -19071.901,E2 -19071.901} C_VEL
LIN {X 0,Y 249.285,Z 517.431,A -85,B 0,C 180,E1 -19075.148,E2 -19075.148} C_VEL
LIN {X 0,Y 249.675,Z 517.382,A -85,B 0,C 180,E1 -19078.387,E2 -19078.387} C_VEL
LIN {X 0,Y 249.672,Z 517.382,A -85,B 0,C 180,E1 -19081.613,E2 -19081.613} C_VEL
LIN {X 0,Y 249.429,Z 517.413,A -85,B 0,C 180,E1 -19086.471,E2 -19086.471} C_VEL
LIN {X 0,Y 249.345,Z 517.423,A -85,B 0,C 180,E1 -19089.736,E2 -19089.736} C_VEL
LIN {X 0,Y 249.184,Z 517.445,A -85,B 0,C 180,E1 -19094.704,E2 -19094.704} C_VEL
LIN {X 0,Y 249.113,Z 517.452,A -85,B 0,C 180,E1 -19098.079,E2 -19098.079} C_VEL
LIN {X 0,Y 249.081,Z 517.454,A -85,B 0,C 180,E1 -19101.518,E2 -19101.518} C_VEL
LIN {X 0,Y 249.087,Z 517.456,A -85,B 0,C 180,E1 -19105.46,E2 -19105.46} C_VEL
LIN {X 0,Y 249.039,Z 517.463,A -85,B 0,C 180,E1 -19108.975,E2 -19108.975} C_VEL
LIN {X 0,Y 249.027,Z 517.468,A -85,B 0,C 180,E1 -19112.426,E2 -19112.426} C_VEL
LIN {X 0,Y 249.048,Z 517.463,A -85,B 0,C 180,E1 -19116.342,E2 -19116.342} C_VEL
LIN {X 0,Y 249.119,Z 517.636,A -85,B 0,C 180,E1 -19118.101,E2 -19118.101} C_VEL
LIN {X 0,Y 250.453,Z 524.668,A -85,B 0,C 180,E1 -19122.335,E2 -19122.335} C_VEL
LIN {X 0,Y 250.954,Z 527.199,A -85,B 0,C 180,E1 -19123.81,E2 -19123.81} C_VEL
LIN {X 0,Y 250.695,Z 529.507,A -85,B 0,C 180,E1 -19125.05,E2 -19125.05} C_VEL
LIN {X 0,Y 248.539,Z 533.581,A -85,B 0,C 180,E1 -19127.068,E2 -19127.068} C_VEL
LIN {X 0,Y 246.419,Z 537.699,A -85,B 0,C 180,E1 -19129.119,E2 -19129.119} C_VEL
LIN {X 0,Y 246.248,Z 540.081,A -85,B 0,C 180,E1 -19130.389,E2 -19130.389} C_VEL
LIN {X 0,Y 246.096,Z 543.375,A -85,B 0,C 180,E1 -19132.121,E2 -19132.121} C_VEL
LIN {X 0,Y 244.211,Z 552.67,A -85,B 0,C 180,E1 -19136.853,E2 -19136.853} C_VEL
LIN {X 0,Y 242.429,Z 563.583,A -85,B 0,C 180,E1 -19142.365,E2 -19142.365} C_VEL
LIN {X 0,Y 242.2,Z 565.121,A -85,B 0,C 180,E1 -19143.14,E2 -19143.14} C_VEL
LIN {X 0,Y 243.431,Z 579.344,A -85,B 0,C 180,E1 -19144.055,E2 -19144.055} C_VEL
LIN {X 0,Y 244.319,Z 592.619,A -85,B 0,C 180,E1 -19145.235,E2 -19145.235} C_VEL
LIN {X 0,Y 244.794,Z 605.672,A -85,B 0,C 180,E1 -19146.739,E2 -19146.739} C_VEL
LIN {X 0,Y 244.975,Z 616.708,A -85,B 0,C 180,E1 -19148.324,E2 -19148.324} C_VEL
LIN {X 0,Y 244.824,Z 627.852,A -85,B 0,C 180,E1 -19150.288,E2 -19150.288} C_VEL
LIN {X 0,Y 244.548,Z 632.048,A -85,B 0,C 180,E1 -19151.137,E2 -19151.137} C_VEL
LIN {X 0,Y 243.196,Z 640.914,A -85,B 0,C 180,E1 -19153.203,E2 -19153.203} C_VEL
LIN {X 0,Y 241.968,Z 649.599,A -85,B 0,C 180,E1 -19155.707,E2 -19155.707} C_VEL
LIN {X 0,Y 241.357,Z 656.556,A -85,B 0,C 180,E1 -19158.239,E2 -19158.239} C_VEL
LIN {X 0,Y 241.149,Z 662.094,A -85,B 0,C 180,E1 -19160.776,E2 -19160.776} C_VEL
LIN {X 0,Y 241.323,Z 666.391,A -85,B 0,C 180,E1 -19163.311,E2 -19163.311} C_VEL
LIN {X 0,Y 241.586,Z 668.62,A -85,B 0,C 180,E1 -19164.993,E2 -19164.993} C_VEL
LIN {X 0,Y 241.746,Z 670.334,A -85,B 0,C 180,E1 -19166.667,E2 -19166.667} C_VEL
LIN {X 0,Y 242.087,Z 671.571,A -85,B 0,C 180,E1 -19168.337,E2 -19168.337} C_VEL
LIN {X 0,Y 242.323,Z 672.351,A -85,B 0,C 180,E1 -19170,E2 -19170} C_VEL
LIN {X 0,Y 241.829,Z 672.584,A -85,B 0,C 180,E1 -19171.666,E2 -19171.666} C_VEL
LIN {X 0,Y 241.508,Z 672.411,A -85,B 0,C 180,E1 -19173.337,E2 -19173.337} C_VEL
LIN {X 0,Y 241.22,Z 671.792,A -85,B 0,C 180,E1 -19175.015,E2 -19175.015} C_VEL
LIN {X 0,Y 240.899,Z 670.331,A -85,B 0,C 180,E1 -19177.29,E2 -19177.29} C_VEL
LIN {X 0,Y 240.797,Z 666.401,A -85,B 0,C 180,E1 -19180.936,E2 -19180.936} C_VEL
LIN {X 0,Y 241.394,Z 662.553,A -85,B 0,C 180,E1 -19183.469,E2 -19183.469} C_VEL
LIN {X 0,Y 242.475,Z 657.69,A -85,B 0,C 180,E1 -19185.983,E2 -19185.983} C_VEL
LIN {X 0,Y 243.709,Z 652.855,A -85,B 0,C 180,E1 -19188.037,E2 -19188.037} C_VEL
LIN {X 0,Y 245.972,Z 645.767,A -85,B 0,C 180,E1 -19190.488,E2 -19190.488} C_VEL
LIN {X 0,Y 248.205,Z 638.856,A -85,B 0,C 180,E1 -19192.474,E2 -19192.474} C_VEL
LIN {X 0,Y 250.406,Z 628.926,A -85,B 0,C 180,E1 -19194.898,E2 -19194.898} C_VEL
LIN {X 0,Y 252.523,Z 618.246,A -85,B 0,C 180,E1 -19197.052,E2 -19197.052} C_VEL
LIN {X 0,Y 253.692,Z 607.335,A -85,B 0,C 180,E1 -19199,E2 -19199} C_VEL
LIN {X 0,Y 253.947,Z 595.492,A -85,B 0,C 180,E1 -19200.916,E2 -19200.916} C_VEL
LIN {X 0,Y 253.161,Z 582.714,A -85,B 0,C 180,E1 -19202.853,E2 -19202.853} C_VEL
LIN {X 0,Y 251.587,Z 571.62,A -85,B 0,C 180,E1 -19204.504,E2 -19204.504} C_VEL
LIN {X 0,Y 249.174,Z 560.48,A -85,B 0,C 180,E1 -19206.194,E2 -19206.194} C_VEL
LIN {X 0,Y 248.033,Z 555.836,A -85,B 0,C 180,E1 -19206.902,E2 -19206.902} C_VEL
LIN {X 0,Y 246.808,Z 551.83,A -85,B 0,C 180,E1 -19207.543,E2 -19207.543} C_VEL
LIN {X 0,Y 246.677,Z 550.539,A -85,B 0,C 180,E1 -19207.71,E2 -19207.71} C_VEL
LIN {X 0,Y 247.466,Z 547.656,A -85,B 0,C 180,E1 -19209.313,E2 -19209.313} C_VEL
LIN {X 0,Y 247.259,Z 544.123,A -85,B 0,C 180,E1 -19211.54,E2 -19211.54} C_VEL
LIN {X 0,Y 246.299,Z 538.457,A -85,B 0,C 180,E1 -19215.51,E2 -19215.51} C_VEL
LIN {X 0,Y 245.229,Z 533.008,A -85,B 0,C 180,E1 -19219.849,E2 -19219.849} C_VEL
LIN {X 0,Y 244.332,Z 528.875,A -85,B 0,C 180,E1 -19223.649,E2 -19223.649} C_VEL
LIN {X 0,Y 243.702,Z 525.914,A -85,B 0,C 180,E1 -19226.775,E2 -19226.775} C_VEL
LIN {X 0,Y 243.069,Z 522.83,A -85,B 0,C 180,E1 -19230.559,E2 -19230.559} C_VEL
LIN {X 0,Y 242.509,Z 520.384,A -85,B 0,C 180,E1 -19234.234,E2 -19234.234} C_VEL
LIN {X 0,Y 242.056,Z 518.326,A -85,B 0,C 180,E1 -19238.298,E2 -19238.298} C_VEL
LIN {X 0,Y 242.166,Z 518.317,A -85,B 0,C 180,E1 -19243.279,E2 -19243.279} C_VEL
LIN {X 0,Y 242.19,Z 518.308,A -85,B 0,C 180,E1 -19248.28,E2 -19248.28} C_VEL
LIN {X 0,Y 242.439,Z 518.277,A -85,B 0,C 180,E1 -19251.666,E2 -19251.666} C_VEL
LIN {X 0,Y 242.25,Z 518.3,A -85,B 0,C 180,E1 -19255.007,E2 -19255.007} C_VEL
LIN {X 0,Y 242.256,Z 518.305,A -85,B 0,C 180,E1 -19255.477,E2 -19255.477} C_VEL
LIN {X 0,Y 243.186,Z 520.95,A -85,B 0,C 180,E1 -19256.117,E2 -19256.117} C_VEL
LIN {X 0,Y 245.382,Z 523.18,A -85,B 0,C 180,E1 -19257.128,E2 -19257.128} C_VEL
LIN {X 0,Y 246.035,Z 524.099,A -85,B 0,C 180,E1 -19257.454,E2 -19257.454} C_VEL
LIN {X 0,Y 247.744,Z 527.017,A -85,B 0,C 180,E1 -19258.375,E2 -19258.375} C_VEL
LIN {X 0,Y 248.637,Z 527.982,A -85,B 0,C 180,E1 -19258.786,E2 -19258.786} C_VEL
LIN {X 0,Y 253.08,Z 536.774,A -85,B 0,C 180,E1 -19261.344,E2 -19261.344} C_VEL
LIN {X 0,Y 257.392,Z 546.96,A -85,B 0,C 180,E1 -19264.207,E2 -19264.207} C_VEL
LIN {X 0,Y 259.86,Z 555.809,A -85,B 0,C 180,E1 -19266.601,E2 -19266.601} C_VEL
LIN {X 0,Y 261.218,Z 562.733,A -85,B 0,C 180,E1 -19268.51,E2 -19268.51} C_VEL
LIN {X 0,Y 260.79,Z 565.403,A -85,B 0,C 180,E1 -19269.11,E2 -19269.11} C_VEL
LIN {X 0,Y 257.901,Z 574.489,A -85,B 0,C 180,E1 -19271.176,E2 -19271.176} C_VEL
LIN {X 0,Y 254.891,Z 582.705,A -85,B 0,C 180,E1 -19273.525,E2 -19273.525} C_VEL
LIN {X 0,Y 252.392,Z 588.886,A -85,B 0,C 180,E1 -19275.754,E2 -19275.754} C_VEL
LIN {X 0,Y 250.23,Z 593.79,A -85,B 0,C 180,E1 -19277.996,E2 -19277.996} C_VEL
LIN {X 0,Y 247.962,Z 598.337,A -85,B 0,C 180,E1 -19280.719,E2 -19280.719} C_VEL
LIN {X 0,Y 245.892,Z 601.853,A -85,B 0,C 180,E1 -19283.848,E2 -19283.848} C_VEL
LIN {X 0,Y 244.359,Z 603.845,A -85,B 0,C 180,E1 -19286.925,E2 -19286.925} C_VEL
LIN {X 0,Y 243.305,Z 604.405,A -85,B 0,C 180,E1 -19289.937,E2 -19289.937} C_VEL
LIN {X 0,Y 242.691,Z 603.697,A -85,B 0,C 180,E1 -19292.88,E2 -19292.88} C_VEL
LIN {X 0,Y 242.462,Z 601.829,A -85,B 0,C 180,E1 -19295.746,E2 -19295.746} C_VEL
LIN {X 0,Y 242.514,Z 598.89,A -85,B 0,C 180,E1 -19298.513,E2 -19298.513} C_VEL
LIN {X 0,Y 243.078,Z 594.001,A -85,B 0,C 180,E1 -19301.682,E2 -19301.682} C_VEL
LIN {X 0,Y 243.913,Z 588.516,A -85,B 0,C 180,E1 -19304.325,E2 -19304.325} C_VEL
LIN {X 0,Y 244.865,Z 582.22,A -85,B 0,C 180,E1 -19306.747,E2 -19306.747} C_VEL
LIN {X 0,Y 246.038,Z 574.649,A -85,B 0,C 180,E1 -19309.115,E2 -19309.115} C_VEL
LIN {X 0,Y 247.506,Z 565.242,A -85,B 0,C 180,E1 -19311.479,E2 -19311.479} C_VEL
LIN {X 0,Y 249.028,Z 554.522,A -85,B 0,C 180,E1 -19313.654,E2 -19313.654} C_VEL
LIN {X 0,Y 249.976,Z 547.507,A -85,B 0,C 180,E1 -19314.83,E2 -19314.83} C_VEL
LIN {X 0,Y 249.564,Z 544.131,A -85,B 0,C 180,E1 -19315.411,E2 -19315.411} C_VEL
LIN {X 0,Y 246.554,Z 533.106,A -85,B 0,C 180,E1 -19317.207,E2 -19317.207} C_VEL
LIN {X 0,Y 242.886,Z 521.301,A -85,B 0,C 180,E1 -19318.854,E2 -19318.854} C_VEL
LIN {X 0,Y 242.012,Z 518.345,A -85,B 0,C 180,E1 -19319.214,E2 -19319.214} C_VEL
LIN {X 0,Y 242.072,Z 518.331,A -85,B 0,C 180,E1 -19324.183,E2 -19324.183} C_VEL
LIN {X 0,Y 242.028,Z 518.335,A -85,B 0,C 180,E1 -19328.315,E2 -19328.315} C_VEL
LIN {X 0,Y 242.132,Z 518.326,A -85,B 0,C 180,E1 -19333.307,E2 -19333.307} C_VEL
LIN {X 0,Y 242.182,Z 518.316,A -85,B 0,C 180,E1 -19338.279,E2 -19338.279} C_VEL
LIN {X 0,Y 242.39,Z 518.292,A -85,B 0,C 180,E1 -19341.664,E2 -19341.664} C_VEL
LIN {X 0,Y 242.25,Z 518.31,A -85,B 0,C 180,E1 -19345.007,E2 -19345.007} C_VEL
LIN {X 0,Y 242.638,Z 518.258,A -85,B 0,C 180,E1 -19348.34,E2 -19348.34} C_VEL
LIN {X 0,Y 242.638,Z 518.26,A -85,B 0,C 180,E1 -19351.66,E2 -19351.66} C_VEL
LIN {X 0,Y 242.403,Z 518.288,A -85,B 0,C 180,E1 -19356.66,E2 -19356.66} C_VEL
LIN {X 0,Y 242.27,Z 518.304,A -85,B 0,C 180,E1 -19360.023,E2 -19360.023} C_VEL
LIN {X 0,Y 242.143,Z 518.324,A -85,B 0,C 180,E1 -19365.142,E2 -19365.142} C_VEL
LIN {X 0,Y 242.064,Z 518.329,A -85,B 0,C 180,E1 -19368.625,E2 -19368.625} C_VEL
LIN {X 0,Y 242.01,Z 518.337,A -85,B 0,C 180,E1 -19372.18,E2 -19372.18} C_VEL
LIN {X 0,Y 242.035,Z 518.332,A -85,B 0,C 180,E1 -19375.821,E2 -19375.821} C_VEL
LIN {X 0,Y 241.974,Z 518.343,A -85,B 0,C 180,E1 -19379.588,E2 -19379.588} C_VEL
LIN {X 0,Y 241.982,Z 518.34,A -85,B 0,C 180,E1 -19383.492,E2 -19383.492} C_VEL
LIN {X 0,Y 241.987,Z 518.341,A -85,B 0,C 180,E1 -19387.582,E2 -19387.582} C_VEL
LIN {X 0,Y 241.926,Z 518.346,A -85,B 0,C 180,E1 -19391.925,E2 -19391.925} C_VEL
LIN {X 0,Y 241.928,Z 518.348,A -85,B 0,C 180,E1 -19396.573,E2 -19396.573} C_VEL
LIN {X 0,Y 241.959,Z 518.342,A -85,B 0,C 180,E1 -19400.28,E2 -19400.28} C_VEL
LIN {X 0,Y 241.99,Z 518.34,A -85,B 0,C 180,E1 -19404.489,E2 -19404.489} C_VEL
LIN {X 0,Y 241.977,Z 518.341,A -85,B 0,C 180,E1 -19408.48,E2 -19408.48} C_VEL
LIN {X 0,Y 242.009,Z 518.336,A -85,B 0,C 180,E1 -19412.312,E2 -19412.312} C_VEL
LIN {X 0,Y 242.044,Z 518.332,A -85,B 0,C 180,E1 -19416.014,E2 -19416.014} C_VEL
LIN {X 0,Y 242.038,Z 518.333,A -85,B 0,C 180,E1 -19419.607,E2 -19419.607} C_VEL
LIN {X 0,Y 242.165,Z 518.32,A -85,B 0,C 180,E1 -19423.278,E2 -19423.278} C_VEL
LIN {X 0,Y 242.182,Z 518.314,A -85,B 0,C 180,E1 -19428.279,E2 -19428.279} C_VEL
LIN {X 0,Y 242.388,Z 518.29,A -85,B 0,C 180,E1 -19431.664,E2 -19431.664} C_VEL
LIN {X 0,Y 242.245,Z 518.309,A -85,B 0,C 180,E1 -19435.006,E2 -19435.006} C_VEL
LIN {X 0,Y 242.635,Z 518.259,A -85,B 0,C 180,E1 -19438.34,E2 -19438.34} C_VEL
LIN {X 0,Y 242.632,Z 518.259,A -85,B 0,C 180,E1 -19441.659,E2 -19441.659} C_VEL
LIN {X 0,Y 242.399,Z 518.29,A -85,B 0,C 180,E1 -19446.659,E2 -19446.659} C_VEL
LIN {X 0,Y 242.269,Z 518.305,A -85,B 0,C 180,E1 -19450.023,E2 -19450.023} C_VEL
LIN {X 0,Y 242.141,Z 518.323,A -85,B 0,C 180,E1 -19455.142,E2 -19455.142} C_VEL
LIN {X 0,Y 242.05,Z 518.335,A -85,B 0,C 180,E1 -19458.626,E2 -19458.626} C_VEL
LIN {X 0,Y 242.004,Z 518.336,A -85,B 0,C 180,E1 -19462.181,E2 -19462.181} C_VEL
LIN {X 0,Y 242.032,Z 518.334,A -85,B 0,C 180,E1 -19465.821,E2 -19465.821} C_VEL
LIN {X 0,Y 241.97,Z 518.342,A -85,B 0,C 180,E1 -19469.588,E2 -19469.588} C_VEL
LIN {X 0,Y 241.979,Z 518.342,A -85,B 0,C 180,E1 -19473.492,E2 -19473.492} C_VEL
LIN {X 0,Y 242.021,Z 518.342,A -85,B 0,C 180,E1 -19477.576,E2 -19477.576} C_VEL
LIN {X 0,Y 243.257,Z 524.852,A -85,B 0,C 180,E1 -19481.644,E2 -19481.644} C_VEL
LIN {X 0,Y 244.679,Z 532.069,A -85,B 0,C 180,E1 -19485.896,E2 -19485.896} C_VEL
LIN {X 0,Y 246.248,Z 540.081,A -85,B 0,C 180,E1 -19490.389,E2 -19490.389} C_VEL
LIN {X 0,Y 246.125,Z 541.654,A -85,B 0,C 180,E1 -19491.219,E2 -19491.219} C_VEL
LIN {X 0,Y 244.671,Z 544.111,A -85,B 0,C 180,E1 -19492.424,E2 -19492.424} C_VEL
LIN {X 0,Y 237.802,Z 551.54,A -85,B 0,C 180,E1 -19496.006,E2 -19496.006} C_VEL
LIN {X 0,Y 237.085,Z 553.226,A -85,B 0,C 180,E1 -19496.875,E2 -19496.875} C_VEL
LIN {X 0,Y 235.252,Z 564.212,A -85,B 0,C 180,E1 -19502.582,E2 -19502.582} C_VEL
LIN {X 0,Y 236.452,Z 578.298,A -85,B 0,C 180,E1 -19503.523,E2 -19503.523} C_VEL
LIN {X 0,Y 237.264,Z 591.02,A -85,B 0,C 180,E1 -19504.681,E2 -19504.681} C_VEL
LIN {X 0,Y 237.751,Z 603.362,A -85,B 0,C 180,E1 -19506.129,E2 -19506.129} C_VEL
LIN {X 0,Y 237.954,Z 615.372,A -85,B 0,C 180,E1 -19507.879,E2 -19507.879} C_VEL
LIN {X 0,Y 237.786,Z 626.624,A -85,B 0,C 180,E1 -19509.905,E2 -19509.905} C_VEL
LIN {X 0,Y 237.474,Z 631.842,A -85,B 0,C 180,E1 -19511.002,E2 -19511.002} C_VEL
LIN {X 0,Y 236.112,Z 640.567,A -85,B 0,C 180,E1 -19513.129,E2 -19513.129} C_VEL
LIN {X 0,Y 235.022,Z 647.779,A -85,B 0,C 180,E1 -19515.275,E2 -19515.275} C_VEL
LIN {X 0,Y 234.379,Z 654.928,A -85,B 0,C 180,E1 -19517.884,E2 -19517.884} C_VEL
LIN {X 0,Y 234.109,Z 660.578,A -85,B 0,C 180,E1 -19520.496,E2 -19520.496} C_VEL
LIN {X 0,Y 234.271,Z 664.982,A -85,B 0,C 180,E1 -19523.108,E2 -19523.108} C_VEL
LIN {X 0,Y 234.54,Z 667.264,A -85,B 0,C 180,E1 -19524.843,E2 -19524.843} C_VEL
LIN {X 0,Y 234.712,Z 669.045,A -85,B 0,C 180,E1 -19526.567,E2 -19526.567} C_VEL
LIN {X 0,Y 235.058,Z 670.362,A -85,B 0,C 180,E1 -19528.287,E2 -19528.287} C_VEL
LIN {X 0,Y 235.298,Z 671.187,A -85,B 0,C 180,E1 -19530,E2 -19530} C_VEL
LIN {X 0,Y 234.446,Z 671.34,A -85,B 0,C 180,E1 -19533.437,E2 -19533.437} C_VEL
LIN {X 0,Y 234.152,Z 670.79,A -85,B 0,C 180,E1 -19535.166,E2 -19535.166} C_VEL
LIN {X 0,Y 233.827,Z 669.507,A -85,B 0,C 180,E1 -19537.315,E2 -19537.315} C_VEL
LIN {X 0,Y 233.665,Z 666.641,A -85,B 0,C 180,E1 -19540.397,E2 -19540.397} C_VEL
LIN {X 0,Y 234.141,Z 663.203,A -85,B 0,C 180,E1 -19543.01,E2 -19543.01} C_VEL
LIN {X 0,Y 235.117,Z 658.785,A -85,B 0,C 180,E1 -19545.606,E2 -19545.606} C_VEL
LIN {X 0,Y 236.611,Z 653.237,A -85,B 0,C 180,E1 -19548.213,E2 -19548.213} C_VEL
LIN {X 0,Y 239.318,Z 645.52,A -85,B 0,C 180,E1 -19551.085,E2 -19551.085} C_VEL
LIN {X 0,Y 241.582,Z 638.739,A -85,B 0,C 180,E1 -19553.125,E2 -19553.125} C_VEL
LIN {X 0,Y 243.934,Z 629.053,A -85,B 0,C 180,E1 -19555.606,E2 -19555.606} C_VEL
LIN {X 0,Y 246.117,Z 619.173,A -85,B 0,C 180,E1 -19557.721,E2 -19557.721} C_VEL
LIN {X 0,Y 247.396,Z 609.444,A -85,B 0,C 180,E1 -19559.577,E2 -19559.577} C_VEL
LIN {X 0,Y 247.967,Z 595.652,A -85,B 0,C 180,E1 -19561.973,E2 -19561.973} C_VEL
LIN {X 0,Y 247.451,Z 583.552,A -85,B 0,C 180,E1 -19563.926,E2 -19563.926} C_VEL
LIN {X 0,Y 245.611,Z 569.984,A -85,B 0,C 180,E1 -19566.105,E2 -19566.105} C_VEL
LIN {X 0,Y 243.407,Z 559.631,A -85,B 0,C 180,E1 -19567.82,E2 -19567.82} C_VEL
LIN {X 0,Y 241.892,Z 553.905,A -85,B 0,C 180,E1 -19568.82,E2 -19568.82} C_VEL
LIN {X 0,Y 240.735,Z 549.781,A -85,B 0,C 180,E1 -19569.538,E2 -19569.538} C_VEL
LIN {X 0,Y 240.569,Z 548.7,A -85,B 0,C 180,E1 -19569.712,E2 -19569.712} C_VEL
LIN {X 0,Y 240.2,Z 544.806,A -85,B 0,C 180,E1 -19572.296,E2 -19572.296} C_VEL
LIN {X 0,Y 239.247,Z 539.313,A -85,B 0,C 180,E1 -19576.346,E2 -19576.346} C_VEL
LIN {X 0,Y 238.393,Z 534.875,A -85,B 0,C 180,E1 -19580.041,E2 -19580.041} C_VEL
LIN {X 0,Y 237.568,Z 530.982,A -85,B 0,C 180,E1 -19583.725,E2 -19583.725} C_VEL
LIN {X 0,Y 236.763,Z 527.374,A -85,B 0,C 180,E1 -19587.703,E2 -19587.703} C_VEL
LIN {X 0,Y 236.172,Z 524.431,A -85,B 0,C 180,E1 -19591.568,E2 -19591.568} C_VEL
LIN {X 0,Y 235.641,Z 522.114,A -85,B 0,C 180,E1 -19595.32,E2 -19595.32} C_VEL
LIN {X 0,Y 235.236,Z 520.325,A -85,B 0,C 180,E1 -19598.991,E2 -19598.991} C_VEL
LIN {X 0,Y 235.071,Z 519.195,A -85,B 0,C 180,E1 -19602.604,E2 -19602.604} C_VEL
LIN {X 0,Y 235.11,Z 519.193,A -85,B 0,C 180,E1 -19606.165,E2 -19606.165} C_VEL
LIN {X 0,Y 235.394,Z 519.155,A -85,B 0,C 180,E1 -19611.415,E2 -19611.415} C_VEL
LIN {X 0,Y 235.381,Z 519.159,A -85,B 0,C 180,E1 -19612.818,E2 -19612.818} C_VEL
LIN {X 0,Y 236.311,Z 521.945,A -85,B 0,C 180,E1 -19613.597,E2 -19613.597} C_VEL
LIN {X 0,Y 238.158,Z 524.046,A -85,B 0,C 180,E1 -19614.603,E2 -19614.603} C_VEL
LIN {X 0,Y 238.873,Z 524.796,A -85,B 0,C 180,E1 -19614.99,E2 -19614.99} C_VEL
LIN {X 0,Y 239.675,Z 526.648,A -85,B 0,C 180,E1 -19615.554,E2 -19615.554} C_VEL
LIN {X 0,Y 242.468,Z 530.267,A -85,B 0,C 180,E1 -19617.101,E2 -19617.101} C_VEL
LIN {X 0,Y 244.673,Z 533.654,A -85,B 0,C 180,E1 -19618.354,E2 -19618.354} C_VEL
LIN {X 0,Y 249.103,Z 543.367,A -85,B 0,C 180,E1 -19621.365,E2 -19621.365} C_VEL
LIN {X 0,Y 252.316,Z 551.917,A -85,B 0,C 180,E1 -19623.942,E2 -19623.942} C_VEL
LIN {X 0,Y 254.342,Z 560.208,A -85,B 0,C 180,E1 -19626.346,E2 -19626.346} C_VEL
LIN {X 0,Y 255.17,Z 565.49,A -85,B 0,C 180,E1 -19627.916,E2 -19627.916} C_VEL
LIN {X 0,Y 254.29,Z 569.144,A -85,B 0,C 180,E1 -19628.744,E2 -19628.744} C_VEL
LIN {X 0,Y 251.167,Z 578.013,A -85,B 0,C 180,E1 -19630.916,E2 -19630.916} C_VEL
LIN {X 0,Y 248.383,Z 585.048,A -85,B 0,C 180,E1 -19633.083,E2 -19633.083} C_VEL
LIN {X 0,Y 245.335,Z 591.881,A -85,B 0,C 180,E1 -19635.792,E2 -19635.792} C_VEL
LIN {X 0,Y 242.677,Z 597.235,A -85,B 0,C 180,E1 -19638.577,E2 -19638.577} C_VEL
LIN {X 0,Y 240.782,Z 600.579,A -85,B 0,C 180,E1 -19640.927,E2 -19640.927} C_VEL
LIN {X 0,Y 238.724,Z 603.669,A -85,B 0,C 180,E1 -19644.126,E2 -19644.126} C_VEL
LIN {X 0,Y 237.201,Z 605.215,A -85,B 0,C 180,E1 -19647.268,E2 -19647.268} C_VEL
LIN {X 0,Y 236.169,Z 605.439,A -85,B 0,C 180,E1 -19650.391,E2 -19650.391} C_VEL
LIN {X 0,Y 235.593,Z 604.439,A -85,B 0,C 180,E1 -19653.355,E2 -19653.355} C_VEL
LIN {X 0,Y 235.409,Z 601.88,A -85,B 0,C 180,E1 -19656.662,E2 -19656.662} C_VEL
LIN {X 0,Y 235.68,Z 597.817,A -85,B 0,C 180,E1 -19659.964,E2 -19659.964} C_VEL
LIN {X 0,Y 236.438,Z 592.239,A -85,B 0,C 180,E1 -19663.132,E2 -19663.132} C_VEL
LIN {X 0,Y 237.392,Z 586.157,A -85,B 0,C 180,E1 -19665.793,E2 -19665.793} C_VEL
LIN {X 0,Y 238.353,Z 579.608,A -85,B 0,C 180,E1 -19668.118,E2 -19668.118} C_VEL
LIN {X 0,Y 239.826,Z 570.911,A -85,B 0,C 180,E1 -19670.617,E2 -19670.617} C_VEL
LIN {X 0,Y 241.379,Z 561.021,A -85,B 0,C 180,E1 -19672.906,E2 -19672.906} C_VEL
LIN {X 0,Y 242.828,Z 550.49,A -85,B 0,C 180,E1 -19674.884,E2 -19674.884} C_VEL
LIN {X 0,Y 243.06,Z 547.215,A -85,B 0,C 180,E1 -19675.427,E2 -19675.427} C_VEL
LIN {X 0,Y 240.305,Z 536.771,A -85,B 0,C 180,E1 -19677.244,E2 -19677.244} C_VEL
LIN {X 0,Y 236.803,Z 525.154,A -85,B 0,C 180,E1 -19678.957,E2 -19678.957} C_VEL
LIN {X 0,Y 234.981,Z 519.22,A -85,B 0,C 180,E1 -19679.739,E2 -19679.739} C_VEL
LIN {X 0,Y 234.999,Z 519.214,A -85,B 0,C 180,E1 -19683.794,E2 -19683.794} C_VEL
LIN {X 0,Y 234.995,Z 519.213,A -85,B 0,C 180,E1 -19688.968,E2 -19688.968} C_VEL
LIN {X 0,Y 235.068,Z 519.205,A -85,B 0,C 180,E1 -19693.086,E2 -19693.086} C_VEL
LIN {X 0,Y 235.115,Z 519.198,A -85,B 0,C 180,E1 -19697.922,E2 -19697.922} C_VEL
LIN {X 0,Y 235.324,Z 519.174,A -85,B 0,C 180,E1 -19701.412,E2 -19701.412} C_VEL
LIN {X 0,Y 235.36,Z 519.168,A -85,B 0,C 180,E1 -19703.14,E2 -19703.14} C_VEL
LIN {X 0,Y 235.598,Z 519.135,A -85,B 0,C 180,E1 -19708.29,E2 -19708.29} C_VEL
LIN {X 0,Y 235.597,Z 519.137,A -85,B 0,C 180,E1 -19711.709,E2 -19711.709} C_VEL
LIN {X 0,Y 235.354,Z 519.167,A -85,B 0,C 180,E1 -19716.86,E2 -19716.86} C_VEL
LIN {X 0,Y 235.216,Z 519.182,A -85,B 0,C 180,E1 -19720.327,E2 -19720.327} C_VEL
LIN {X 0,Y 235.097,Z 519.198,A -85,B 0,C 180,E1 -19725.607,E2 -19725.607} C_VEL
LIN {X 0,Y 235.004,Z 519.212,A -85,B 0,C 180,E1 -19729.206,E2 -19729.206} C_VEL
LIN {X 0,Y 234.955,Z 519.218,A -85,B 0,C 180,E1 -19732.883,E2 -19732.883} C_VEL
LIN {X 0,Y 234.95,Z 519.215,A -85,B 0,C 180,E1 -19736.66,E2 -19736.66} C_VEL
LIN {X 0,Y 234.903,Z 519.223,A -85,B 0,C 180,E1 -19740.572,E2 -19740.572} C_VEL
LIN {X 0,Y 234.929,Z 519.217,A -85,B 0,C 180,E1 -19744.638,E2 -19744.638} C_VEL
LIN {X 0,Y 234.914,Z 519.224,A -85,B 0,C 180,E1 -19748.935,E2 -19748.935} C_VEL
LIN {X 0,Y 234.876,Z 519.226,A -85,B 0,C 180,E1 -19753.489,E2 -19753.489} C_VEL
LIN {X 0,Y 234.881,Z 519.226,A -85,B 0,C 180,E1 -19756.512,E2 -19756.512} C_VEL
LIN {X 0,Y 234.921,Z 519.221,A -85,B 0,C 180,E1 -19761.078,E2 -19761.078} C_VEL
LIN {X 0,Y 234.933,Z 519.221,A -85,B 0,C 180,E1 -19765.362,E2 -19765.362} C_VEL
LIN {X 0,Y 234.934,Z 519.217,A -85,B 0,C 180,E1 -19769.432,E2 -19769.432} C_VEL
LIN {X 0,Y 234.996,Z 519.211,A -85,B 0,C 180,E1 -19773.793,E2 -19773.793} C_VEL
LIN {X 0,Y 235,Z 519.211,A -85,B 0,C 180,E1 -19778.968,E2 -19778.968} C_VEL
LIN {X 0,Y 235.099,Z 519.202,A -85,B 0,C 180,E1 -19783.059,E2 -19783.059} C_VEL
LIN {X 0,Y 235.116,Z 519.193,A -85,B 0,C 180,E1 -19787.922,E2 -19787.922} C_VEL
LIN {X 0,Y 235.322,Z 519.171,A -85,B 0,C 180,E1 -19791.412,E2 -19791.412} C_VEL
LIN {X 0,Y 235.359,Z 519.167,A -85,B 0,C 180,E1 -19793.14,E2 -19793.14} C_VEL
LIN {X 0,Y 235.595,Z 519.136,A -85,B 0,C 180,E1 -19798.29,E2 -19798.29} C_VEL
LIN {X 0,Y 235.591,Z 519.136,A -85,B 0,C 180,E1 -19801.709,E2 -19801.709} C_VEL
LIN {X 0,Y 235.35,Z 519.169,A -85,B 0,C 180,E1 -19806.86,E2 -19806.86} C_VEL
LIN {X 0,Y 235.215,Z 519.184,A -85,B 0,C 180,E1 -19810.327,E2 -19810.327} C_VEL
LIN {X 0,Y 235.087,Z 519.199,A -85,B 0,C 180,E1 -19815.608,E2 -19815.608} C_VEL
LIN {X 0,Y 234.991,Z 519.212,A -85,B 0,C 180,E1 -19819.207,E2 -19819.207} C_VEL
LIN {X 0,Y 234.947,Z 519.219,A -85,B 0,C 180,E1 -19822.884,E2 -19822.884} C_VEL
LIN {X 0,Y 234.946,Z 519.22,A -85,B 0,C 180,E1 -19826.66,E2 -19826.66} C_VEL
LIN {X 0,Y 234.899,Z 519.225,A -85,B 0,C 180,E1 -19830.572,E2 -19830.572} C_VEL
LIN {X 0,Y 234.93,Z 519.223,A -85,B 0,C 180,E1 -19834.638,E2 -19834.638} C_VEL
LIN {X 0,Y 234.982,Z 519.361,A -85,B 0,C 180,E1 -19837.275,E2 -19837.275} C_VEL
LIN {X 0,Y 236.395,Z 526.756,A -85,B 0,C 180,E1 -19841.991,E2 -19841.991} C_VEL
LIN {X 0,Y 237.787,Z 533.794,A -85,B 0,C 180,E1 -19846.246,E2 -19846.246} C_VEL
LIN {X 0,Y 239.01,Z 540.041,A -85,B 0,C 180,E1 -19849.864,E2 -19849.864} C_VEL
LIN {X 0,Y 239.275,Z 541.942,A -85,B 0,C 180,E1 -19850.924,E2 -19850.924} C_VEL
LIN {X 0,Y 238.487,Z 546.315,A -85,B 0,C 180,E1 -19853.238,E2 -19853.238} C_VEL
LIN {X 0,Y 237.085,Z 553.226,A -85,B 0,C 180,E1 -19856.875,E2 -19856.875} C_VEL
LIN {X 0,Y 236.079,Z 554.874,A -85,B 0,C 180,E1 -19857.715,E2 -19857.715} C_VEL
LIN {X 0,Y 232.767,Z 557.473,A -85,B 0,C 180,E1 -19858.998,E2 -19858.998} C_VEL
LIN {X 0,Y 229.468,Z 560.07,A -85,B 0,C 180,E1 -19860.314,E2 -19860.314} C_VEL
LIN {X 0,Y 228.513,Z 561.727,A -85,B 0,C 180,E1 -19861.193,E2 -19861.193} C_VEL
LIN {X 0,Y 228.298,Z 563.166,A -85,B 0,C 180,E1 -19861.97,E2 -19861.97} C_VEL
LIN {X 0,Y 229.537,Z 578.221,A -85,B 0,C 180,E1 -19863.034,E2 -19863.034} C_VEL
LIN {X 0,Y 230.338,Z 591.335,A -85,B 0,C 180,E1 -19864.309,E2 -19864.309} C_VEL
LIN {X 0,Y 230.769,Z 604.972,A -85,B 0,C 180,E1 -19866.013,E2 -19866.013} C_VEL
LIN {X 0,Y 230.901,Z 616.737,A -85,B 0,C 180,E1 -19867.873,E2 -19867.873} C_VEL
LIN {X 0,Y 230.695,Z 627.524,A -85,B 0,C 180,E1 -19869.957,E2 -19869.957} C_VEL
LIN {X 0,Y 230.168,Z 632.994,A -85,B 0,C 180,E1 -19871.184,E2 -19871.184} C_VEL
LIN {X 0,Y 228.775,Z 641.687,A -85,B 0,C 180,E1 -19873.491,E2 -19873.491} C_VEL
LIN {X 0,Y 227.735,Z 649.792,A -85,B 0,C 180,E1 -19876.163,E2 -19876.163} C_VEL
LIN {X 0,Y 227.256,Z 655.307,A -85,B 0,C 180,E1 -19878.404,E2 -19878.404} C_VEL
LIN {X 0,Y 227.075,Z 660.66,A -85,B 0,C 180,E1 -19881.098,E2 -19881.098} C_VEL
LIN {X 0,Y 227.331,Z 664.787,A -85,B 0,C 180,E1 -19883.788,E2 -19883.788} C_VEL
LIN {X 0,Y 227.676,Z 667.74,A -85,B 0,C 180,E1 -19886.461,E2 -19886.461} C_VEL
LIN {X 0,Y 228.027,Z 669.141,A -85,B 0,C 180,E1 -19888.234,E2 -19888.234} C_VEL
LIN {X 0,Y 228.272,Z 670.023,A -85,B 0,C 180,E1 -19890,E2 -19890} C_VEL
LIN {X 0,Y 227.385,Z 670.253,A -85,B 0,C 180,E1 -19893.544,E2 -19893.544} C_VEL
LIN {X 0,Y 227.084,Z 669.766,A -85,B 0,C 180,E1 -19895.328,E2 -19895.328} C_VEL
LIN {X 0,Y 226.768,Z 668.678,A -85,B 0,C 180,E1 -19897.368,E2 -19897.368} C_VEL
LIN {X 0,Y 226.64,Z 665.786,A -85,B 0,C 180,E1 -19900.723,E2 -19900.723} C_VEL
LIN {X 0,Y 227.465,Z 661.161,A -85,B 0,C 180,E1 -19904.311,E2 -19904.311} C_VEL
LIN {X 0,Y 228.676,Z 656.548,A -85,B 0,C 180,E1 -19906.976,E2 -19906.976} C_VEL
LIN {X 0,Y 229.807,Z 652.871,A -85,B 0,C 180,E1 -19908.73,E2 -19908.73} C_VEL
LIN {X 0,Y 232.226,Z 646.408,A -85,B 0,C 180,E1 -19911.295,E2 -19911.295} C_VEL
LIN {X 0,Y 235.012,Z 638.609,A -85,B 0,C 180,E1 -19913.811,E2 -19913.811} C_VEL
LIN {X 0,Y 237.508,Z 629.284,A -85,B 0,C 180,E1 -19916.351,E2 -19916.351} C_VEL
LIN {X 0,Y 239.917,Z 619.108,A -85,B 0,C 180,E1 -19918.641,E2 -19918.641} C_VEL
LIN {X 0,Y 241.451,Z 607.977,A -85,B 0,C 180,E1 -19920.865,E2 -19920.865} C_VEL
LIN {X 0,Y 242.095,Z 595.87,A -85,B 0,C 180,E1 -19923.079,E2 -19923.079} C_VEL
LIN {X 0,Y 241.68,Z 583.677,A -85,B 0,C 180,E1 -19925.201,E2 -19925.201} C_VEL
LIN {X 0,Y 240.473,Z 572.843,A -85,B 0,C 180,E1 -19927.07,E2 -19927.07} C_VEL
LIN {X 0,Y 238.592,Z 562.624,A -85,B 0,C 180,E1 -19928.909,E2 -19928.909} C_VEL
LIN {X 0,Y 237.542,Z 557.833,A -85,B 0,C 180,E1 -19929.797,E2 -19929.797} C_VEL
LIN {X 0,Y 236.323,Z 553.239,A -85,B 0,C 180,E1 -19930.683,E2 -19930.683} C_VEL
LIN {X 0,Y 233.856,Z 548.244,A -85,B 0,C 180,E1 -19932.093,E2 -19932.093} C_VEL
LIN {X 0,Y 233.284,Z 546.203,A -85,B 0,C 180,E1 -19932.59,E2 -19932.59} C_VEL
LIN {X 0,Y 232.392,Z 541.042,A -85,B 0,C 180,E1 -19936.537,E2 -19936.537} C_VEL
LIN {X 0,Y 231.523,Z 536.564,A -85,B 0,C 180,E1 -19940.397,E2 -19940.397} C_VEL
LIN {X 0,Y 231.092,Z 534.314,A -85,B 0,C 180,E1 -19942.538,E2 -19942.538} C_VEL
LIN {X 0,Y 230.222,Z 530.504,A -85,B 0,C 180,E1 -19946.668,E2 -19946.668} C_VEL
LIN {X 0,Y 229.561,Z 527.37,A -85,B 0,C 180,E1 -19950.67,E2 -19950.67} C_VEL
LIN {X 0,Y 229.02,Z 524.895,A -85,B 0,C 180,E1 -19954.557,E2 -19954.557} C_VEL
LIN {X 0,Y 228.599,Z 522.971,A -85,B 0,C 180,E1 -19958.351,E2 -19958.351} C_VEL
LIN {X 0,Y 228.311,Z 521.346,A -85,B 0,C 180,E1 -19962.605,E2 -19962.605} C_VEL
LIN {X 0,Y 228.134,Z 520.09,A -85,B 0,C 180,E1 -19967.999,E2 -19967.999} C_VEL
LIN {X 0,Y 228.2,Z 520.174,A -85,B 0,C 180,E1 -19969.388,E2 -19969.388} C_VEL
LIN {X 0,Y 229.014,Z 522.384,A -85,B 0,C 180,E1 -19970.159,E2 -19970.159} C_VEL
LIN {X 0,Y 231.077,Z 524.784,A -85,B 0,C 180,E1 -19971.584,E2 -19971.584} C_VEL
LIN {X 0,Y 232.334,Z 525.854,A -85,B 0,C 180,E1 -19972.341,E2 -19972.341} C_VEL
LIN {X 0,Y 233.51,Z 528.543,A -85,B 0,C 180,E1 -19973.322,E2 -19973.322} C_VEL
LIN {X 0,Y 235.272,Z 530.442,A -85,B 0,C 180,E1 -19974.386,E2 -19974.386} C_VEL
LIN {X 0,Y 236.768,Z 533.349,A -85,B 0,C 180,E1 -19975.467,E2 -19975.467} C_VEL
LIN {X 0,Y 239.26,Z 537.176,A -85,B 0,C 180,E1 -19977.101,E2 -19977.101} C_VEL
LIN {X 0,Y 241.078,Z 540.443,A -85,B 0,C 180,E1 -19978.33,E2 -19978.33} C_VEL
LIN {X 0,Y 244.641,Z 549.217,A -85,B 0,C 180,E1 -19981.236,E2 -19981.236} C_VEL
LIN {X 0,Y 247.124,Z 556.731,A -85,B 0,C 180,E1 -19983.669,E2 -19983.669} C_VEL
LIN {X 0,Y 248.721,Z 564.497,A -85,B 0,C 180,E1 -19986.083,E2 -19986.083} C_VEL
LIN {X 0,Y 249.214,Z 568.296,A -85,B 0,C 180,E1 -19987.292,E2 -19987.292} C_VEL
LIN {X 0,Y 246.168,Z 577.132,A -85,B 0,C 180,E1 -19989.449,E2 -19989.449} C_VEL
LIN {X 0,Y 243.084,Z 584.63,A -85,B 0,C 180,E1 -19991.677,E2 -19991.677} C_VEL
LIN {X 0,Y 239.919,Z 591.521,A -85,B 0,C 180,E1 -19994.278,E2 -19994.278} C_VEL
LIN {X 0,Y 236.827,Z 597.441,A -85,B 0,C 180,E1 -19997.263,E2 -19997.263} C_VEL
LIN {X 0,Y 234.344,Z 601.604,A -85,B 0,C 180,E1 -20000.169,E2 -20000.169} C_VEL
LIN {X 0,Y 232.277,Z 604.531,A -85,B 0,C 180,E1 -20003.163,E2 -20003.163} C_VEL
LIN {X 0,Y 231.142,Z 605.757,A -85,B 0,C 180,E1 -20005.194,E2 -20005.194} C_VEL
LIN {X 0,Y 230.031,Z 606.539,A -85,B 0,C 180,E1 -20007.622,E2 -20007.622} C_VEL
LIN {X 0,Y 229.038,Z 606.39,A -85,B 0,C 180,E1 -20010.775,E2 -20010.775} C_VEL
LIN {X 0,Y 228.526,Z 605.037,A -85,B 0,C 180,E1 -20013.865,E2 -20013.865} C_VEL
LIN {X 0,Y 228.365,Z 602.584,A -85,B 0,C 180,E1 -20016.854,E2 -20016.854} C_VEL
LIN {X 0,Y 228.66,Z 598.393,A -85,B 0,C 180,E1 -20020.2,E2 -20020.2} C_VEL
LIN {X 0,Y 229.223,Z 594.316,A -85,B 0,C 180,E1 -20022.621,E2 -20022.621} C_VEL
LIN {X 0,Y 230.151,Z 588.412,A -85,B 0,C 180,E1 -20025.384,E2 -20025.384} C_VEL
LIN {X 0,Y 231.213,Z 581.365,A -85,B 0,C 180,E1 -20028.031,E2 -20028.031} C_VEL
LIN {X 0,Y 232.7,Z 572.746,A -85,B 0,C 180,E1 -20030.636,E2 -20030.636} C_VEL
LIN {X 0,Y 234.316,Z 562.877,A -85,B 0,C 180,E1 -20033.021,E2 -20033.021} C_VEL
LIN {X 0,Y 235.929,Z 551.582,A -85,B 0,C 180,E1 -20035.228,E2 -20035.228} C_VEL
LIN {X 0,Y 236.241,Z 549.447,A -85,B 0,C 180,E1 -20035.581,E2 -20035.581} C_VEL
LIN {X 0,Y 233.651,Z 539.005,A -85,B 0,C 180,E1 -20037.475,E2 -20037.475} C_VEL
LIN {X 0,Y 230.53,Z 528.398,A -85,B 0,C 180,E1 -20039.147,E2 -20039.147} C_VEL
LIN {X 0,Y 227.961,Z 520.093,A -85,B 0,C 180,E1 -20040.298,E2 -20040.298} C_VEL
LIN {X 0,Y 227.93,Z 520.093,A -85,B 0,C 180,E1 -20044.426,E2 -20044.426} C_VEL
LIN {X 0,Y 227.949,Z 520.089,A -85,B 0,C 180,E1 -20048.285,E2 -20048.285} C_VEL
LIN {X 0,Y 228.013,Z 520.083,A -85,B 0,C 180,E1 -20052.847,E2 -20052.847} C_VEL
LIN {X 0,Y 228.071,Z 520.077,A -85,B 0,C 180,E1 -20057.543,E2 -20057.543} C_VEL
LIN {X 0,Y 228.262,Z 520.053,A -85,B 0,C 180,E1 -20061.144,E2 -20061.144} C_VEL
LIN {X 0,Y 228.313,Z 520.045,A -85,B 0,C 180,E1 -20062.927,E2 -20062.927} C_VEL
LIN {X 0,Y 228.556,Z 520.013,A -85,B 0,C 180,E1 -20068.238,E2 -20068.238} C_VEL
LIN {X 0,Y 228.555,Z 520.013,A -85,B 0,C 180,E1 -20071.762,E2 -20071.762} C_VEL
LIN {X 0,Y 228.306,Z 520.046,A -85,B 0,C 180,E1 -20077.073,E2 -20077.073} C_VEL
LIN {X 0,Y 228.146,Z 520.063,A -85,B 0,C 180,E1 -20080.651,E2 -20080.651} C_VEL
LIN {X 0,Y 228.047,Z 520.074,A -85,B 0,C 180,E1 -20086.103,E2 -20086.103} C_VEL
LIN {X 0,Y 227.936,Z 520.09,A -85,B 0,C 180,E1 -20089.826,E2 -20089.826} C_VEL
LIN {X 0,Y 227.903,Z 520.094,A -85,B 0,C 180,E1 -20093.634,E2 -20093.634} C_VEL
LIN {X 0,Y 227.861,Z 520.1,A -85,B 0,C 180,E1 -20097.558,E2 -20097.558} C_VEL
LIN {X 0,Y 227.859,Z 520.1,A -85,B 0,C 180,E1 -20101.624,E2 -20101.624} C_VEL
LIN {X 0,Y 227.882,Z 520.096,A -85,B 0,C 180,E1 -20105.871,E2 -20105.871} C_VEL
LIN {X 0,Y 227.809,Z 520.106,A -85,B 0,C 180,E1 -20110.38,E2 -20110.38} C_VEL
LIN {X 0,Y 227.827,Z 520.107,A -85,B 0,C 180,E1 -20115.194,E2 -20115.194} C_VEL
LIN {X 0,Y 227.827,Z 520.103,A -85,B 0,C 180,E1 -20119.623,E2 -20119.623} C_VEL
LIN {X 0,Y 227.883,Z 520.096,A -85,B 0,C 180,E1 -20124.128,E2 -20124.128} C_VEL
LIN {X 0,Y 227.873,Z 520.098,A -85,B 0,C 180,E1 -20128.377,E2 -20128.377} C_VEL
LIN {X 0,Y 227.888,Z 520.096,A -85,B 0,C 180,E1 -20132.445,E2 -20132.445} C_VEL
LIN {X 0,Y 227.909,Z 520.094,A -85,B 0,C 180,E1 -20136.366,E2 -20136.366} C_VEL
LIN {X 0,Y 227.94,Z 520.088,A -85,B 0,C 180,E1 -20140.174,E2 -20140.174} C_VEL
LIN {X 0,Y 228.06,Z 520.075,A -85,B 0,C 180,E1 -20143.897,E2 -20143.897} C_VEL
LIN {X 0,Y 228.074,Z 520.071,A -85,B 0,C 180,E1 -20147.543,E2 -20147.543} C_VEL
LIN {X 0,Y 228.26,Z 520.053,A -85,B 0,C 180,E1 -20151.144,E2 -20151.144} C_VEL
LIN {X 0,Y 228.311,Z 520.047,A -85,B 0,C 180,E1 -20152.927,E2 -20152.927} C_VEL
LIN {X 0,Y 228.553,Z 520.013,A -85,B 0,C 180,E1 -20158.237,E2 -20158.237} C_VEL
LIN {X 0,Y 228.549,Z 520.013,A -85,B 0,C 180,E1 -20161.762,E2 -20161.762} C_VEL
LIN {X 0,Y 228.303,Z 520.047,A -85,B 0,C 180,E1 -20167.073,E2 -20167.073} C_VEL
LIN {X 0,Y 228.146,Z 520.066,A -85,B 0,C 180,E1 -20170.651,E2 -20170.651} C_VEL
LIN {X 0,Y 228.05,Z 520.075,A -85,B 0,C 180,E1 -20174.273,E2 -20174.273} C_VEL
LIN {X 0,Y 227.969,Z 520.086,A -85,B 0,C 180,E1 -20177.956,E2 -20177.956} C_VEL
LIN {X 0,Y 227.921,Z 520.09,A -85,B 0,C 180,E1 -20182.323,E2 -20182.323} C_VEL
LIN {X 0,Y 227.923,Z 520.095,A -85,B 0,C 180,E1 -20186.592,E2 -20186.592} C_VEL
LIN {X 0,Y 227.874,Z 520.098,A -85,B 0,C 180,E1 -20190.281,E2 -20190.281} C_VEL
LIN {X 0,Y 227.877,Z 520.099,A -85,B 0,C 180,E1 -20193.72,E2 -20193.72} C_VEL
LIN {X 0,Y 227.949,Z 520.188,A -85,B 0,C 180,E1 -20196.824,E2 -20196.824} C_VEL
LIN {X 0,Y 229.218,Z 526.846,A -85,B 0,C 180,E1 -20201.239,E2 -20201.239} C_VEL
LIN {X 0,Y 230.518,Z 533.609,A -85,B 0,C 180,E1 -20205.475,E2 -20205.475} C_VEL
LIN {X 0,Y 231.984,Z 541.04,A -85,B 0,C 180,E1 -20209.918,E2 -20209.918} C_VEL
LIN {X 0,Y 232.114,Z 543.584,A -85,B 0,C 180,E1 -20211.353,E2 -20211.353} C_VEL
LIN {X 0,Y 230.309,Z 552.139,A -85,B 0,C 180,E1 -20216.017,E2 -20216.017} C_VEL
LIN {X 0,Y 228.513,Z 561.727,A -85,B 0,C 180,E1 -20221.193,E2 -20221.193} C_VEL
LIN {X 0,Y 228.343,Z 563.36,A -85,B 0,C 180,E1 -20221.691,E2 -20221.691} C_VEL
LIN {X 0,Y 228.082,Z 567.319,A -85,B 0,C 180,E1 -20222.182,E2 -20222.182} C_VEL
LIN {X 0,Y 227.075,Z 576.045,A -85,B 0,C 180,E1 -20222.686,E2 -20222.686} C_VEL
LIN {X 0,Y 223.76,Z 587.39,A -85,B 0,C 180,E1 -20223.461,E2 -20223.461} C_VEL
LIN {X 0,Y 223.376,Z 591.056,A -85,B 0,C 180,E1 -20223.862,E2 -20223.862} C_VEL
LIN {X 0,Y 223.762,Z 603.447,A -85,B 0,C 180,E1 -20225.46,E2 -20225.46} C_VEL
LIN {X 0,Y 223.882,Z 615.383,A -85,B 0,C 180,E1 -20227.385,E2 -20227.385} C_VEL
LIN {X 0,Y 223.638,Z 626.224,A -85,B 0,C 180,E1 -20229.537,E2 -20229.537} C_VEL
LIN {X 0,Y 223.328,Z 631.489,A -85,B 0,C 180,E1 -20230.749,E2 -20230.749} C_VEL
LIN {X 0,Y 221.967,Z 639.776,A -85,B 0,C 180,E1 -20232.97,E2 -20232.97} C_VEL
LIN {X 0,Y 220.779,Z 648.014,A -85,B 0,C 180,E1 -20235.718,E2 -20235.718} C_VEL
LIN {X 0,Y 220.265,Z 653.661,A -85,B 0,C 180,E1 -20238.03,E2 -20238.03} C_VEL
LIN {X 0,Y 220.038,Z 659.126,A -85,B 0,C 180,E1 -20240.811,E2 -20240.811} C_VEL
LIN {X 0,Y 220.265,Z 663.36,A -85,B 0,C 180,E1 -20243.588,E2 -20243.588} C_VEL
LIN {X 0,Y 220.638,Z 666.419,A -85,B 0,C 180,E1 -20246.348,E2 -20246.348} C_VEL
LIN {X 0,Y 220.996,Z 667.87,A -85,B 0,C 180,E1 -20248.178,E2 -20248.178} C_VEL
LIN {X 0,Y 221.249,Z 668.841,A -85,B 0,C 180,E1 -20250,E2 -20250} C_VEL
LIN {X 0,Y 220.74,Z 669.204,A -85,B 0,C 180,E1 -20251.825,E2 -20251.825} C_VEL
LIN {X 0,Y 220.324,Z 669.163,A -85,B 0,C 180,E1 -20253.658,E2 -20253.658} C_VEL
LIN {X 0,Y 220.018,Z 668.721,A -85,B 0,C 180,E1 -20255.499,E2 -20255.499} C_VEL
LIN {X 0,Y 219.697,Z 667.844,A -85,B 0,C 180,E1 -20257.399,E2 -20257.399} C_VEL
LIN {X 0,Y 219.595,Z 664.942,A -85,B 0,C 180,E1 -20261.071,E2 -20261.071} C_VEL
LIN {X 0,Y 220.522,Z 660.459,A -85,B 0,C 180,E1 -20264.771,E2 -20264.771} C_VEL
LIN {X 0,Y 221.818,Z 655.959,A -85,B 0,C 180,E1 -20267.518,E2 -20267.518} C_VEL
LIN {X 0,Y 224.338,Z 649.434,A -85,B 0,C 180,E1 -20270.637,E2 -20270.637} C_VEL
LIN {X 0,Y 227.574,Z 641.243,A -85,B 0,C 180,E1 -20273.67,E2 -20273.67} C_VEL
LIN {X 0,Y 230.201,Z 632.681,A -85,B 0,C 180,E1 -20276.276,E2 -20276.276} C_VEL
LIN {X 0,Y 233.042,Z 622.433,A -85,B 0,C 180,E1 -20278.851,E2 -20278.851} C_VEL
LIN {X 0,Y 234.972,Z 612.348,A -85,B 0,C 180,E1 -20281.061,E2 -20281.061} C_VEL
LIN {X 0,Y 236.193,Z 599.652,A -85,B 0,C 180,E1 -20283.577,E2 -20283.577} C_VEL
LIN {X 0,Y 236.336,Z 588.53,A -85,B 0,C 180,E1 -20285.671,E2 -20285.671} C_VEL
LIN {X 0,Y 235.467,Z 576.338,A -85,B 0,C 180,E1 -20287.935,E2 -20287.935} C_VEL
LIN {X 0,Y 234.142,Z 567.056,A -85,B 0,C 180,E1 -20289.719,E2 -20289.719} C_VEL
LIN {X 0,Y 232.363,Z 558.133,A -85,B 0,C 180,E1 -20291.528,E2 -20291.528} C_VEL
LIN {X 0,Y 230.149,Z 552.97,A -85,B 0,C 180,E1 -20293.028,E2 -20293.028} C_VEL
LIN {X 0,Y 229.548,Z 551.441,A -85,B 0,C 180,E1 -20293.46,E2 -20293.46} C_VEL
LIN {X 0,Y 226.627,Z 546.278,A -85,B 0,C 180,E1 -20295.422,E2 -20295.422} C_VEL
LIN {X 0,Y 225.601,Z 543.232,A -85,B 0,C 180,E1 -20296.356,E2 -20296.356} C_VEL
LIN {X 0,Y 224.788,Z 538.93,A -85,B 0,C 180,E1 -20300.139,E2 -20300.139} C_VEL
LIN {X 0,Y 223.852,Z 534.433,A -85,B 0,C 180,E1 -20304.716,E2 -20304.716} C_VEL
LIN {X 0,Y 222.947,Z 530.378,A -85,B 0,C 180,E1 -20309.711,E2 -20309.711} C_VEL
LIN {X 0,Y 222.405,Z 527.71,A -85,B 0,C 180,E1 -20313.743,E2 -20313.743} C_VEL
LIN {X 0,Y 221.964,Z 525.646,A -85,B 0,C 180,E1 -20317.67,E2 -20317.67} C_VEL
LIN {X 0,Y 221.672,Z 523.904,A -85,B 0,C 180,E1 -20322.016,E2 -20322.016} C_VEL
LIN {X 0,Y 221.499,Z 523.137,A -85,B 0,C 180,E1 -20325.361,E2 -20325.361} C_VEL
LIN {X 0,Y 223.058,Z 525.305,A -85,B 0,C 180,E1 -20326.957,E2 -20326.957} C_VEL
LIN {X 0,Y 225.54,Z 526.857,A -85,B 0,C 180,E1 -20328.884,E2 -20328.884} C_VEL
LIN {X 0,Y 227.073,Z 529.925,A -85,B 0,C 180,E1 -20330.365,E2 -20330.365} C_VEL
LIN {X 0,Y 229.36,Z 532.675,A -85,B 0,C 180,E1 -20332.075,E2 -20332.075} C_VEL
LIN {X 0,Y 230.41,Z 534.786,A -85,B 0,C 180,E1 -20332.992,E2 -20332.992} C_VEL
LIN {X 0,Y 231.591,Z 536.247,A -85,B 0,C 180,E1 -20333.835,E2 -20333.835} C_VEL
LIN {X 0,Y 236.396,Z 544.903,A -85,B 0,C 180,E1 -20337.588,E2 -20337.588} C_VEL
LIN {X 0,Y 239.348,Z 552.873,A -85,B 0,C 180,E1 -20340.421,E2 -20340.421} C_VEL
LIN {X 0,Y 241.423,Z 559.512,A -85,B 0,C 180,E1 -20342.734,E2 -20342.734} C_VEL
LIN {X 0,Y 242.847,Z 567.426,A -85,B 0,C 180,E1 -20345.397,E2 -20345.397} C_VEL
LIN {X 0,Y 243.228,Z 571.103,A -85,B 0,C 180,E1 -20346.637,E2 -20346.637} C_VEL
LIN {X 0,Y 239.965,Z 579.719,A -85,B 0,C 180,E1 -20348.845,E2 -20348.845} C_VEL
LIN {X 0,Y 236.497,Z 587.404,A -85,B 0,C 180,E1 -20351.283,E2 -20351.283} C_VEL
LIN {X 0,Y 233.223,Z 593.878,A -85,B 0,C 180,E1 -20353.95,E2 -20353.95} C_VEL
LIN {X 0,Y 230.157,Z 599.268,A -85,B 0,C 180,E1 -20356.864,E2 -20356.864} C_VEL
LIN {X 0,Y 227.536,Z 603.278,A -85,B 0,C 180,E1 -20359.863,E2 -20359.863} C_VEL
LIN {X 0,Y 226.066,Z 605.185,A -85,B 0,C 180,E1 -20361.905,E2 -20361.905} C_VEL
LIN {X 0,Y 224.351,Z 606.928,A -85,B 0,C 180,E1 -20364.707,E2 -20364.707} C_VEL
LIN {X 0,Y 222.786,Z 607.752,A -85,B 0,C 180,E1 -20368.242,E2 -20368.242} C_VEL
LIN {X 0,Y 221.924,Z 607.266,A -85,B 0,C 180,E1 -20371.234,E2 -20371.234} C_VEL
LIN {X 0,Y 221.415,Z 605.236,A -85,B 0,C 180,E1 -20374.845,E2 -20374.845} C_VEL
LIN {X 0,Y 221.407,Z 601.805,A -85,B 0,C 180,E1 -20378.342,E2 -20378.342} C_VEL
LIN {X 0,Y 221.919,Z 596.961,A -85,B 0,C 180,E1 -20381.687,E2 -20381.687} C_VEL
LIN {X 0,Y 222.774,Z 591.498,A -85,B 0,C 180,E1 -20384.544,E2 -20384.544} C_VEL
LIN {X 0,Y 223.929,Z 584.289,A -85,B 0,C 180,E1 -20387.524,E2 -20387.524} C_VEL
LIN {X 0,Y 225.298,Z 576.077,A -85,B 0,C 180,E1 -20390.209,E2 -20390.209} C_VEL
LIN {X 0,Y 226.9,Z 566.673,A -85,B 0,C 180,E1 -20392.695,E2 -20392.695} C_VEL
LIN {X 0,Y 228.505,Z 556.187,A -85,B 0,C 180,E1 -20394.936,E2 -20394.936} C_VEL
LIN {X 0,Y 229.262,Z 551.07,A -85,B 0,C 180,E1 -20395.863,E2 -20395.863} C_VEL
LIN {X 0,Y 228.51,Z 547.02,A -85,B 0,C 180,E1 -20396.649,E2 -20396.649} C_VEL
LIN {X 0,Y 225.328,Z 535.364,A -85,B 0,C 180,E1 -20398.727,E2 -20398.727} C_VEL
LIN {X 0,Y 222.033,Z 524.659,A -85,B 0,C 180,E1 -20400.358,E2 -20400.358} C_VEL
LIN {X 0,Y 220.893,Z 521.006,A -85,B 0,C 180,E1 -20400.844,E2 -20400.844} C_VEL
LIN {X 0,Y 220.899,Z 520.972,A -85,B 0,C 180,E1 -20403.55,E2 -20403.55} C_VEL
LIN {X 0,Y 220.869,Z 520.974,A -85,B 0,C 180,E1 -20407.552,E2 -20407.552} C_VEL
LIN {X 0,Y 220.967,Z 520.96,A -85,B 0,C 180,E1 -20412.589,E2 -20412.589} C_VEL
LIN {X 0,Y 221.009,Z 520.957,A -85,B 0,C 180,E1 -20417.138,E2 -20417.138} C_VEL
LIN {X 0,Y 221.202,Z 520.931,A -85,B 0,C 180,E1 -20420.859,E2 -20420.859} C_VEL
LIN {X 0,Y 221.132,Z 520.938,A -85,B 0,C 180,E1 -20424.529,E2 -20424.529} C_VEL
LIN {X 0,Y 221.514,Z 520.89,A -85,B 0,C 180,E1 -20428.182,E2 -20428.182} C_VEL
LIN {X 0,Y 221.513,Z 520.891,A -85,B 0,C 180,E1 -20431.818,E2 -20431.818} C_VEL
LIN {X 0,Y 221.244,Z 520.925,A -85,B 0,C 180,E1 -20437.3,E2 -20437.3} C_VEL
LIN {X 0,Y 221.067,Z 520.947,A -85,B 0,C 180,E1 -20440.996,E2 -20440.996} C_VEL
LIN {X 0,Y 221.011,Z 520.952,A -85,B 0,C 180,E1 -20446.63,E2 -20446.63} C_VEL
LIN {X 0,Y 220.888,Z 520.968,A -85,B 0,C 180,E1 -20450.486,E2 -20450.486} C_VEL
LIN {X 0,Y 220.855,Z 520.971,A -85,B 0,C 180,E1 -20454.436,E2 -20454.436} C_VEL
LIN {X 0,Y 220.809,Z 520.978,A -85,B 0,C 180,E1 -20458.517,E2 -20458.517} C_VEL
LIN {X 0,Y 220.815,Z 520.978,A -85,B 0,C 180,E1 -20462.756,E2 -20462.756} C_VEL
LIN {X 0,Y 220.812,Z 520.981,A -85,B 0,C 180,E1 -20467.277,E2 -20467.277} C_VEL
LIN {X 0,Y 220.761,Z 520.982,A -85,B 0,C 180,E1 -20471.955,E2 -20471.955} C_VEL
LIN {X 0,Y 220.769,Z 520.984,A -85,B 0,C 180,E1 -20475.544,E2 -20475.544} C_VEL
LIN {X 0,Y 220.809,Z 520.977,A -85,B 0,C 180,E1 -20480.463,E2 -20480.463} C_VEL
LIN {X 0,Y 220.804,Z 520.982,A -85,B 0,C 180,E1 -20485.045,E2 -20485.045} C_VEL
LIN {X 0,Y 220.87,Z 520.969,A -85,B 0,C 180,E1 -20489.394,E2 -20489.394} C_VEL
LIN {X 0,Y 220.897,Z 520.968,A -85,B 0,C 180,E1 -20493.549,E2 -20493.549} C_VEL
